LIN {X 0,Y 420.578,Z 342.697,A -85,B 0,C 180,E1 -10184.764,E2 -10184.764} C_VEL
LIN {X 0,Y 421.368,Z 331.394,A -85,B 0,C 180,E1 -10185.603,E2 -10185.603} C_VEL
LIN {X 0,Y 422.106,Z 318.707,A -85,B 0,C 180,E1 -10186.319,E2 -10186.319} C_VEL
LIN {X 0,Y 422.68,Z 306.29,A -85,B 0,C 180,E1 -10186.824,E2 -10186.824} C_VEL
LIN {X 0,Y 423.128,Z 292.678,A -85,B 0,C 180,E1 -10187.179,E2 -10187.179} C_VEL
LIN {X 0,Y 424.249,Z 215.121,A -85,B 0,C 180,E1 -10188.698,E2 -10188.698} C_VEL
LIN {X 0,Y 420.632,Z 193.799,A -85,B 0,C 180,E1 -10189.35,E2 -10189.35} C_VEL
LIN {X 0,Y 419.974,Z 190.079,A -85,B 0,C 180,E1 -10189.487,E2 -10189.487} C_VEL
LIN {X 0,Y 421.119,Z 172.26,A -85,B 0,C 180,E1 -10193.004,E2 -10193.004} C_VEL
LIN {X 0,Y 421.346,Z 166.733,A -85,B 0,C 180,E1 -10194.121,E2 -10194.121} C_VEL
LIN {X 0,Y 419.386,Z 156.606,A -85,B 0,C 180,E1 -10196.365,E2 -10196.365} C_VEL
LIN {X 0,Y 418.209,Z 151.397,A -85,B 0,C 180,E1 -10197.595,E2 -10197.595} C_VEL
LIN {X 0,Y 418.236,Z 151.388,A -85,B 0,C 180,E1 -10200.274,E2 -10200.274} C_VEL
LIN {X 0,Y 418.234,Z 151.388,A -85,B 0,C 180,E1 -10203.679,E2 -10203.679} C_VEL
LIN {X 0,Y 418.236,Z 151.388,A -85,B 0,C 180,E1 -10207.225,E2 -10207.225} C_VEL
LIN {X 0,Y 418.209,Z 151.393,A -85,B 0,C 180,E1 -10210.868,E2 -10210.868} C_VEL
LIN {X 0,Y 418.205,Z 151.387,A -85,B 0,C 180,E1 -10213.729,E2 -10213.729} C_VEL
LIN {X 0,Y 418.203,Z 151.387,A -85,B 0,C 180,E1 -10216.448,E2 -10216.448} C_VEL
LIN {X 0,Y 418.209,Z 151.387,A -85,B 0,C 180,E1 -10219.133,E2 -10219.133} C_VEL
LIN {X 0,Y 418.239,Z 151.388,A -85,B 0,C 180,E1 -10222.776,E2 -10222.776} C_VEL
LIN {X 0,Y 418.236,Z 151.387,A -85,B 0,C 180,E1 -10226.322,E2 -10226.322} C_VEL
LIN {X 0,Y 418.241,Z 151.382,A -85,B 0,C 180,E1 -10229.728,E2 -10229.728} C_VEL
LIN {X 0,Y 418.213,Z 151.388,A -85,B 0,C 180,E1 -10233.017,E2 -10233.017} C_VEL
LIN {X 0,Y 418.262,Z 151.384,A -85,B 0,C 180,E1 -10236.217,E2 -10236.217} C_VEL
LIN {X 0,Y 418.253,Z 151.38,A -85,B 0,C 180,E1 -10239.337,E2 -10239.337} C_VEL
LIN {X 0,Y 418.259,Z 151.387,A -85,B 0,C 180,E1 -10242.395,E2 -10242.395} C_VEL
LIN {X 0,Y 418.283,Z 151.382,A -85,B 0,C 180,E1 -10245.402,E2 -10245.402} C_VEL
LIN {X 0,Y 418.317,Z 151.379,A -85,B 0,C 180,E1 -10248.369,E2 -10248.369} C_VEL
LIN {X 0,Y 418.45,Z 151.364,A -85,B 0,C 180,E1 -10252.278,E2 -10252.278} C_VEL
LIN {X 0,Y 418.488,Z 151.359,A -85,B 0,C 180,E1 -10254.217,E2 -10254.217} C_VEL
LIN {X 0,Y 418.538,Z 151.353,A -85,B 0,C 180,E1 -10258.076,E2 -10258.076} C_VEL
LIN {X 0,Y 418.567,Z 151.351,A -85,B 0,C 180,E1 -10260,E2 -10260} C_VEL
LIN {X 0,Y 418.494,Z 151.36,A -85,B 0,C 180,E1 -10262.888,E2 -10262.888} C_VEL
LIN {X 0,Y 418.322,Z 151.452,A -85,B 0,C 180,E1 -10264.396,E2 -10264.396} C_VEL
LIN {X 0,Y 420.077,Z 159.254,A -85,B 0,C 180,E1 -10266.243,E2 -10266.243} C_VEL
LIN {X 0,Y 420.765,Z 163.432,A -85,B 0,C 180,E1 -10267.197,E2 -10267.197} C_VEL
LIN {X 0,Y 420.544,Z 170.284,A -85,B 0,C 180,E1 -10268.62,E2 -10268.62} C_VEL
LIN {X 0,Y 424.721,Z 189.71,A -85,B 0,C 180,E1 -10269.272,E2 -10269.272} C_VEL
LIN {X 0,Y 423.098,Z 278.42,A -85,B 0,C 180,E1 -10271.027,E2 -10271.027} C_VEL
LIN {X 0,Y 422.665,Z 291.77,A -85,B 0,C 180,E1 -10271.483,E2 -10271.483} C_VEL
LIN {X 0,Y 422.127,Z 303.733,A -85,B 0,C 180,E1 -10272.073,E2 -10272.073} C_VEL
LIN {X 0,Y 421.492,Z 315.941,A -85,B 0,C 180,E1 -10272.887,E2 -10272.887} C_VEL
LIN {X 0,Y 420.728,Z 327.426,A -85,B 0,C 180,E1 -10273.867,E2 -10273.867} C_VEL
LIN {X 0,Y 419.975,Z 337.256,A -85,B 0,C 180,E1 -10274.91,E2 -10274.91} C_VEL
LIN {X 0,Y 419.33,Z 346.043,A -85,B 0,C 180,E1 -10276.054,E2 -10276.054} C_VEL
LIN {X 0,Y 418.676,Z 354.422,A -85,B 0,C 180,E1 -10277.39,E2 -10277.39} C_VEL
LIN {X 0,Y 418.137,Z 361.95,A -85,B 0,C 180,E1 -10278.873,E2 -10278.873} C_VEL
LIN {X 0,Y 417.715,Z 367.293,A -85,B 0,C 180,E1 -10280.177,E2 -10280.177} C_VEL
LIN {X 0,Y 417.418,Z 372.376,A -85,B 0,C 180,E1 -10281.741,E2 -10281.741} C_VEL
LIN {X 0,Y 417.206,Z 376.186,A -85,B 0,C 180,E1 -10283.32,E2 -10283.32} C_VEL
LIN {X 0,Y 416.984,Z 378.805,A -85,B 0,C 180,E1 -10284.921,E2 -10284.921} C_VEL
LIN {X 0,Y 416.845,Z 380.338,A -85,B 0,C 180,E1 -10286.672,E2 -10286.672} C_VEL
LIN {X 0,Y 416.858,Z 380.431,A -85,B 0,C 180,E1 -10288.753,E2 -10288.753} C_VEL
LIN {X 0,Y 416.972,Z 378.732,A -85,B 0,C 180,E1 -10290.727,E2 -10290.727} C_VEL
LIN {X 0,Y 417.085,Z 376.61,A -85,B 0,C 180,E1 -10292.046,E2 -10292.046} C_VEL
LIN {X 0,Y 417.236,Z 372.609,A -85,B 0,C 180,E1 -10293.77,E2 -10293.77} C_VEL
LIN {X 0,Y 417.524,Z 366.971,A -85,B 0,C 180,E1 -10295.502,E2 -10295.502} C_VEL
LIN {X 0,Y 417.854,Z 360.816,A -85,B 0,C 180,E1 -10296.963,E2 -10296.963} C_VEL
LIN {X 0,Y 418.368,Z 353.097,A -85,B 0,C 180,E1 -10298.43,E2 -10298.43} C_VEL
LIN {X 0,Y 418.92,Z 344.378,A -85,B 0,C 180,E1 -10299.763,E2 -10299.763} C_VEL
LIN {X 0,Y 419.513,Z 333.739,A -85,B 0,C 180,E1 -10301.072,E2 -10301.072} C_VEL
LIN {X 0,Y 420.165,Z 323.007,A -85,B 0,C 180,E1 -10302.129,E2 -10302.129} C_VEL
LIN {X 0,Y 420.845,Z 311.186,A -85,B 0,C 180,E1 -10303.044,E2 -10303.044} C_VEL
LIN {X 0,Y 421.385,Z 298.499,A -85,B 0,C 180,E1 -10303.801,E2 -10303.801} C_VEL
LIN {X 0,Y 421.825,Z 285.338,A -85,B 0,C 180,E1 -10304.359,E2 -10304.359} C_VEL
LIN {X 0,Y 422.202,Z 272.242,A -85,B 0,C 180,E1 -10304.714,E2 -10304.714} C_VEL
LIN {X 0,Y 423.374,Z 189.479,A -85,B 0,C 180,E1 -10306.269,E2 -10306.269} C_VEL
LIN {X 0,Y 419.77,Z 169.472,A -85,B 0,C 180,E1 -10306.836,E2 -10306.836} C_VEL
LIN {X 0,Y 420.098,Z 162.133,A -85,B 0,C 180,E1 -10308.499,E2 -10308.499} C_VEL
LIN {X 0,Y 418.696,Z 153.617,A -85,B 0,C 180,E1 -10310.546,E2 -10310.546} C_VEL
LIN {X 0,Y 418.278,Z 151.384,A -85,B 0,C 180,E1 -10311.098,E2 -10311.098} C_VEL
LIN {X 0,Y 418.246,Z 151.387,A -85,B 0,C 180,E1 -10313.975,E2 -10313.975} C_VEL
LIN {X 0,Y 418.254,Z 151.382,A -85,B 0,C 180,E1 -10317.158,E2 -10317.158} C_VEL
LIN {X 0,Y 418.26,Z 151.383,A -85,B 0,C 180,E1 -10320.837,E2 -10320.837} C_VEL
LIN {X 0,Y 418.216,Z 151.39,A -85,B 0,C 180,E1 -10324.092,E2 -10324.092} C_VEL
LIN {X 0,Y 418.237,Z 151.385,A -85,B 0,C 180,E1 -10325.759,E2 -10325.759} C_VEL
LIN {X 0,Y 417.607,Z 151.468,A -85,B 0,C 180,E1 -10326.562,E2 -10326.562} C_VEL
LIN {X 0,Y 414.834,Z 151.81,A -85,B 0,C 180,E1 -10327.868,E2 -10327.868} C_VEL
LIN {X 0,Y 412.43,Z 152.108,A -85,B 0,C 180,E1 -10328.922,E2 -10328.922} C_VEL
LIN {X 0,Y 411.333,Z 152.246,A -85,B 0,C 180,E1 -10329.736,E2 -10329.736} C_VEL
LIN {X 0,Y 411.209,Z 152.264,A -85,B 0,C 180,E1 -10330.012,E2 -10330.012} C_VEL
LIN {X 0,Y 411.224,Z 152.257,A -85,B 0,C 180,E1 -10333.151,E2 -10333.151} C_VEL
LIN {X 0,Y 411.311,Z 152.247,A -85,B 0,C 180,E1 -10336.896,E2 -10336.896} C_VEL
LIN {X 0,Y 411.281,Z 152.255,A -85,B 0,C 180,E1 -10340.16,E2 -10340.16} C_VEL
LIN {X 0,Y 411.395,Z 152.236,A -85,B 0,C 180,E1 -10343.131,E2 -10343.131} C_VEL
LIN {X 0,Y 411.289,Z 152.249,A -85,B 0,C 180,E1 -10345.098,E2 -10345.098} C_VEL
LIN {X 0,Y 411.506,Z 152.227,A -85,B 0,C 180,E1 -10348.042,E2 -10348.042} C_VEL
LIN {X 0,Y 411.38,Z 152.238,A -85,B 0,C 180,E1 -10350.978,E2 -10350.978} C_VEL
LIN {X 0,Y 411.431,Z 152.232,A -85,B 0,C 180,E1 -10352.937,E2 -10352.937} C_VEL
LIN {X 0,Y 411.391,Z 152.237,A -85,B 0,C 180,E1 -10356.867,E2 -10356.867} C_VEL
LIN {X 0,Y 411.279,Z 152.255,A -85,B 0,C 180,E1 -10359.838,E2 -10359.838} C_VEL
LIN {X 0,Y 411.308,Z 152.249,A -85,B 0,C 180,E1 -10363.102,E2 -10363.102} C_VEL
LIN {X 0,Y 411.209,Z 152.26,A -85,B 0,C 180,E1 -10366.89,E2 -10366.89} C_VEL
LIN {X 0,Y 411.205,Z 152.261,A -85,B 0,C 180,E1 -10369.987,E2 -10369.987} C_VEL
LIN {X 0,Y 411.188,Z 152.267,A -85,B 0,C 180,E1 -10373.147,E2 -10373.147} C_VEL
LIN {X 0,Y 411.172,Z 152.264,A -85,B 0,C 180,E1 -10376.384,E2 -10376.384} C_VEL
LIN {X 0,Y 411.194,Z 152.263,A -85,B 0,C 180,E1 -10379.712,E2 -10379.712} C_VEL
LIN {X 0,Y 411.203,Z 152.267,A -85,B 0,C 180,E1 -10383.155,E2 -10383.155} C_VEL
LIN {X 0,Y 411.19,Z 152.263,A -85,B 0,C 180,E1 -10386.551,E2 -10386.551} C_VEL
LIN {X 0,Y 411.175,Z 152.264,A -85,B 0,C 180,E1 -10389.721,E2 -10389.721} C_VEL
LIN {X 0,Y 411.159,Z 152.27,A -85,B 0,C 180,E1 -10393.134,E2 -10393.134} C_VEL
LIN {X 0,Y 411.16,Z 152.265,A -85,B 0,C 180,E1 -10395.881,E2 -10395.881} C_VEL
LIN {X 0,Y 411.154,Z 152.266,A -85,B 0,C 180,E1 -10399.492,E2 -10399.492} C_VEL
LIN {X 0,Y 411.179,Z 152.263,A -85,B 0,C 180,E1 -10402.024,E2 -10402.024} C_VEL
LIN {X 0,Y 411.198,Z 152.263,A -85,B 0,C 180,E1 -10405.122,E2 -10405.122} C_VEL
LIN {X 0,Y 411.158,Z 152.267,A -85,B 0,C 180,E1 -10408.002,E2 -10408.002} C_VEL
LIN {X 0,Y 411.165,Z 152.265,A -85,B 0,C 180,E1 -10411.406,E2 -10411.406} C_VEL
LIN {X 0,Y 411.182,Z 152.264,A -85,B 0,C 180,E1 -10414.94,E2 -10414.94} C_VEL
LIN {X 0,Y 411.195,Z 152.263,A -85,B 0,C 180,E1 -10417.913,E2 -10417.913} C_VEL
LIN {X 0,Y 411.207,Z 152.26,A -85,B 0,C 180,E1 -10421.05,E2 -10421.05} C_VEL
LIN {X 0,Y 411.203,Z 152.265,A -85,B 0,C 180,E1 -10424.129,E2 -10424.129} C_VEL
LIN {X 0,Y 411.295,Z 152.248,A -85,B 0,C 180,E1 -10427.165,E2 -10427.165} C_VEL
LIN {X 0,Y 411.268,Z 152.259,A -85,B 0,C 180,E1 -10430.16,E2 -10430.16} C_VEL
LIN {X 0,Y 411.383,Z 152.237,A -85,B 0,C 180,E1 -10433.131,E2 -10433.131} C_VEL
LIN {X 0,Y 411.281,Z 152.25,A -85,B 0,C 180,E1 -10435.098,E2 -10435.098} C_VEL
LIN {X 0,Y 411.494,Z 152.23,A -85,B 0,C 180,E1 -10438.042,E2 -10438.042} C_VEL
LIN {X 0,Y 411.368,Z 152.239,A -85,B 0,C 180,E1 -10440.979,E2 -10440.979} C_VEL
LIN {X 0,Y 411.419,Z 152.233,A -85,B 0,C 180,E1 -10442.937,E2 -10442.937} C_VEL
LIN {X 0,Y 411.419,Z 152.239,A -85,B 0,C 180,E1 -10445.883,E2 -10445.883} C_VEL
LIN {X 0,Y 411.298,Z 152.248,A -85,B 0,C 180,E1 -10448.846,E2 -10448.846} C_VEL
LIN {X 0,Y 411.266,Z 152.257,A -85,B 0,C 180,E1 -10451.833,E2 -10451.833} C_VEL
LIN {X 0,Y 411.221,Z 152.258,A -85,B 0,C 180,E1 -10454.854,E2 -10454.854} C_VEL
LIN {X 0,Y 411.17,Z 152.267,A -85,B 0,C 180,E1 -10457.919,E2 -10457.919} C_VEL
LIN {X 0,Y 411.178,Z 152.265,A -85,B 0,C 180,E1 -10461.035,E2 -10461.035} C_VEL
LIN {X 0,Y 411.18,Z 152.263,A -85,B 0,C 180,E1 -10464.218,E2 -10464.218} C_VEL
LIN {X 0,Y 411.136,Z 152.274,A -85,B 0,C 180,E1 -10467.486,E2 -10467.486} C_VEL
LIN {X 0,Y 411.185,Z 152.265,A -85,B 0,C 180,E1 -10469.714,E2 -10469.714} C_VEL
LIN {X 0,Y 411.197,Z 152.267,A -85,B 0,C 180,E1 -10473.157,E2 -10473.157} C_VEL
LIN {X 0,Y 411.182,Z 152.263,A -85,B 0,C 180,E1 -10476.552,E2 -10476.552} C_VEL
LIN {X 0,Y 411.161,Z 152.266,A -85,B 0,C 180,E1 -10479.721,E2 -10479.721} C_VEL
LIN {X 0,Y 411.155,Z 152.272,A -85,B 0,C 180,E1 -10483.136,E2 -10483.136} C_VEL
LIN {X 0,Y 411.158,Z 152.265,A -85,B 0,C 180,E1 -10485.883,E2 -10485.883} C_VEL
LIN {X 0,Y 411.153,Z 152.267,A -85,B 0,C 180,E1 -10489.494,E2 -10489.494} C_VEL
LIN {X 0,Y 411.176,Z 152.263,A -85,B 0,C 180,E1 -10492.026,E2 -10492.026} C_VEL
LIN {X 0,Y 411.197,Z 152.264,A -85,B 0,C 180,E1 -10495.124,E2 -10495.124} C_VEL
LIN {X 0,Y 411.155,Z 152.266,A -85,B 0,C 180,E1 -10498.003,E2 -10498.003} C_VEL
LIN {X 0,Y 411.165,Z 152.267,A -85,B 0,C 180,E1 -10501.407,E2 -10501.407} C_VEL
LIN {X 0,Y 411.203,Z 152.471,A -85,B 0,C 180,E1 -10502.716,E2 -10502.716} C_VEL
LIN {X 0,Y 413.85,Z 165.762,A -85,B 0,C 180,E1 -10505.682,E2 -10505.682} C_VEL
LIN {X 0,Y 413.938,Z 170.108,A -85,B 0,C 180,E1 -10506.593,E2 -10506.593} C_VEL
LIN {X 0,Y 413.243,Z 180.993,A -85,B 0,C 180,E1 -10508.815,E2 -10508.815} C_VEL
LIN {X 0,Y 412.56,Z 191.635,A -85,B 0,C 180,E1 -10510.923,E2 -10510.923} C_VEL
LIN {X 0,Y 416.315,Z 216.844,A -85,B 0,C 180,E1 -10511.579,E2 -10511.579} C_VEL
LIN {X 0,Y 415.097,Z 300.369,A -85,B 0,C 180,E1 -10513.21,E2 -10513.21} C_VEL
LIN {X 0,Y 414.541,Z 314.458,A -85,B 0,C 180,E1 -10513.693,E2 -10513.693} C_VEL
LIN {X 0,Y 413.983,Z 326.514,A -85,B 0,C 180,E1 -10514.303,E2 -10514.303} C_VEL
LIN {X 0,Y 413.303,Z 338.276,A -85,B 0,C 180,E1 -10515.097,E2 -10515.097} C_VEL
LIN {X 0,Y 412.61,Z 349.81,A -85,B 0,C 180,E1 -10516.092,E2 -10516.092} C_VEL
LIN {X 0,Y 411.954,Z 359.966,A -85,B 0,C 180,E1 -10517.187,E2 -10517.187} C_VEL
LIN {X 0,Y 411.366,Z 369.225,A -85,B 0,C 180,E1 -10518.42,E2 -10518.42} C_VEL
LIN {X 0,Y 410.821,Z 378.248,A -85,B 0,C 180,E1 -10519.902,E2 -10519.902} C_VEL
LIN {X 0,Y 410.422,Z 385.465,A -85,B 0,C 180,E1 -10521.384,E2 -10521.384} C_VEL
LIN {X 0,Y 410.162,Z 392.029,A -85,B 0,C 180,E1 -10523.112,E2 -10523.112} C_VEL
LIN {X 0,Y 410.011,Z 396.332,A -85,B 0,C 180,E1 -10524.591,E2 -10524.591} C_VEL
LIN {X 0,Y 409.931,Z 399.529,A -85,B 0,C 180,E1 -10526.069,E2 -10526.069} C_VEL
LIN {X 0,Y 409.928,Z 401.113,A -85,B 0,C 180,E1 -10527.053,E2 -10527.053} C_VEL
LIN {X 0,Y 409.966,Z 402.238,A -85,B 0,C 180,E1 -10528.036,E2 -10528.036} C_VEL
LIN {X 0,Y 409.936,Z 402.929,A -85,B 0,C 180,E1 -10529.019,E2 -10529.019} C_VEL
LIN {X 0,Y 409.928,Z 403.22,A -85,B 0,C 180,E1 -10530.001,E2 -10530.001} C_VEL
LIN {X 0,Y 409.936,Z 403.108,A -85,B 0,C 180,E1 -10530.983,E2 -10530.983} C_VEL
LIN {X 0,Y 409.966,Z 402.547,A -85,B 0,C 180,E1 -10531.966,E2 -10531.966} C_VEL
LIN {X 0,Y 409.924,Z 401.57,A -85,B 0,C 180,E1 -10532.949,E2 -10532.949} C_VEL
LIN {X 0,Y 409.931,Z 400.185,A -85,B 0,C 180,E1 -10533.933,E2 -10533.933} C_VEL
LIN {X 0,Y 410.013,Z 397.264,A -85,B 0,C 180,E1 -10535.41,E2 -10535.41} C_VEL
LIN {X 0,Y 410.167,Z 393.284,A -85,B 0,C 180,E1 -10536.89,E2 -10536.89} C_VEL
LIN {X 0,Y 410.467,Z 387.179,A -85,B 0,C 180,E1 -10538.617,E2 -10538.617} C_VEL
LIN {X 0,Y 410.9,Z 380.464,A -85,B 0,C 180,E1 -10540.098,E2 -10540.098} C_VEL
LIN {X 0,Y 411.501,Z 372.131,A -85,B 0,C 180,E1 -10541.577,E2 -10541.577} C_VEL
LIN {X 0,Y 412.262,Z 363.629,A -85,B 0,C 180,E1 -10542.805,E2 -10542.805} C_VEL
LIN {X 0,Y 412.924,Z 353.201,A -85,B 0,C 180,E1 -10544.035,E2 -10544.035} C_VEL
LIN {X 0,Y 413.849,Z 341.458,A -85,B 0,C 180,E1 -10545.136,E2 -10545.136} C_VEL
LIN {X 0,Y 414.691,Z 329.881,A -85,B 0,C 180,E1 -10545.987,E2 -10545.987} C_VEL
LIN {X 0,Y 415.443,Z 316.74,A -85,B 0,C 180,E1 -10546.714,E2 -10546.714} C_VEL
LIN {X 0,Y 416.1,Z 303.661,A -85,B 0,C 180,E1 -10547.225,E2 -10547.225} C_VEL
LIN {X 0,Y 416.513,Z 288.254,A -85,B 0,C 180,E1 -10547.587,E2 -10547.587} C_VEL
LIN {X 0,Y 417.662,Z 216.047,A -85,B 0,C 180,E1 -10549.042,E2 -10549.042} C_VEL
LIN {X 0,Y 413.962,Z 194.236,A -85,B 0,C 180,E1 -10549.727,E2 -10549.727} C_VEL
LIN {X 0,Y 413.153,Z 189.85,A -85,B 0,C 180,E1 -10549.891,E2 -10549.891} C_VEL
LIN {X 0,Y 414.318,Z 172.758,A -85,B 0,C 180,E1 -10553.335,E2 -10553.335} C_VEL
LIN {X 0,Y 414.465,Z 168.182,A -85,B 0,C 180,E1 -10554.281,E2 -10554.281} C_VEL
LIN {X 0,Y 412.487,Z 158.086,A -85,B 0,C 180,E1 -10556.568,E2 -10556.568} C_VEL
LIN {X 0,Y 411.167,Z 152.272,A -85,B 0,C 180,E1 -10557.969,E2 -10557.969} C_VEL
LIN {X 0,Y 411.186,Z 152.269,A -85,B 0,C 180,E1 -10560.849,E2 -10560.849} C_VEL
LIN {X 0,Y 411.194,Z 152.264,A -85,B 0,C 180,E1 -10564.335,E2 -10564.335} C_VEL
LIN {X 0,Y 411.188,Z 152.268,A -85,B 0,C 180,E1 -10566.743,E2 -10566.743} C_VEL
LIN {X 0,Y 411.17,Z 152.267,A -85,B 0,C 180,E1 -10569.721,E2 -10569.721} C_VEL
LIN {X 0,Y 411.165,Z 152.267,A -85,B 0,C 180,E1 -10573.136,E2 -10573.136} C_VEL
LIN {X 0,Y 411.167,Z 152.262,A -85,B 0,C 180,E1 -10575.882,E2 -10575.882} C_VEL
LIN {X 0,Y 411.161,Z 152.264,A -85,B 0,C 180,E1 -10579.493,E2 -10579.493} C_VEL
LIN {X 0,Y 411.187,Z 152.261,A -85,B 0,C 180,E1 -10582.025,E2 -10582.025} C_VEL
LIN {X 0,Y 411.206,Z 152.263,A -85,B 0,C 180,E1 -10585.124,E2 -10585.124} C_VEL
LIN {X 0,Y 411.167,Z 152.268,A -85,B 0,C 180,E1 -10588.003,E2 -10588.003} C_VEL
LIN {X 0,Y 411.174,Z 152.263,A -85,B 0,C 180,E1 -10591.407,E2 -10591.407} C_VEL
LIN {X 0,Y 411.191,Z 152.263,A -85,B 0,C 180,E1 -10594.942,E2 -10594.942} C_VEL
LIN {X 0,Y 411.207,Z 152.262,A -85,B 0,C 180,E1 -10597.914,E2 -10597.914} C_VEL
LIN {X 0,Y 411.218,Z 152.259,A -85,B 0,C 180,E1 -10601.051,E2 -10601.051} C_VEL
LIN {X 0,Y 411.215,Z 152.262,A -85,B 0,C 180,E1 -10604.13,E2 -10604.13} C_VEL
LIN {X 0,Y 411.308,Z 152.251,A -85,B 0,C 180,E1 -10607.166,E2 -10607.166} C_VEL
LIN {X 0,Y 411.292,Z 152.255,A -85,B 0,C 180,E1 -10610.161,E2 -10610.161} C_VEL
LIN {X 0,Y 411.394,Z 152.242,A -85,B 0,C 180,E1 -10613.132,E2 -10613.132} C_VEL
LIN {X 0,Y 411.294,Z 152.253,A -85,B 0,C 180,E1 -10615.099,E2 -10615.099} C_VEL
LIN {X 0,Y 411.506,Z 152.229,A -85,B 0,C 180,E1 -10618.043,E2 -10618.043} C_VEL
LIN {X 0,Y 411.519,Z 152.229,A -85,B 0,C 180,E1 -10620,E2 -10620} C_VEL
LIN {X 0,Y 411.451,Z 152.238,A -85,B 0,C 180,E1 -10622.938,E2 -10622.938} C_VEL
LIN {X 0,Y 411.285,Z 152.396,A -85,B 0,C 180,E1 -10624.042,E2 -10624.042} C_VEL
LIN {X 0,Y 413.244,Z 160.916,A -85,B 0,C 180,E1 -10626.102,E2 -10626.102} C_VEL
LIN {X 0,Y 413.947,Z 166.194,A -85,B 0,C 180,E1 -10627.316,E2 -10627.316} C_VEL
LIN {X 0,Y 413.696,Z 170.425,A -85,B 0,C 180,E1 -10628.211,E2 -10628.211} C_VEL
LIN {X 0,Y 417.966,Z 189.659,A -85,B 0,C 180,E1 -10628.887,E2 -10628.887} C_VEL
LIN {X 0,Y 418.143,Z 194.672,A -85,B 0,C 180,E1 -10629.005,E2 -10629.005} C_VEL
LIN {X 0,Y 416.403,Z 279.017,A -85,B 0,C 180,E1 -10630.718,E2 -10630.718} C_VEL
LIN {X 0,Y 415.943,Z 291.904,A -85,B 0,C 180,E1 -10631.169,E2 -10631.169} C_VEL
LIN {X 0,Y 415.373,Z 304.045,A -85,B 0,C 180,E1 -10631.777,E2 -10631.777} C_VEL
LIN {X 0,Y 414.713,Z 316.222,A -85,B 0,C 180,E1 -10632.603,E2 -10632.603} C_VEL
LIN {X 0,Y 413.893,Z 327.999,A -85,B 0,C 180,E1 -10633.627,E2 -10633.627} C_VEL
LIN {X 0,Y 413.035,Z 338.568,A -85,B 0,C 180,E1 -10634.788,E2 -10634.788} C_VEL
LIN {X 0,Y 412.291,Z 348.029,A -85,B 0,C 180,E1 -10636.082,E2 -10636.082} C_VEL
LIN {X 0,Y 411.633,Z 356.12,A -85,B 0,C 180,E1 -10637.44,E2 -10637.44} C_VEL
LIN {X 0,Y 411.03,Z 363.399,A -85,B 0,C 180,E1 -10638.958,E2 -10638.958} C_VEL
LIN {X 0,Y 410.584,Z 369.364,A -85,B 0,C 180,E1 -10640.543,E2 -10640.543} C_VEL
LIN {X 0,Y 410.248,Z 374.442,A -85,B 0,C 180,E1 -10642.318,E2 -10642.318} C_VEL
LIN {X 0,Y 410.14,Z 376.405,A -85,B 0,C 180,E1 -10643.211,E2 -10643.211} C_VEL
LIN {X 0,Y 409.938,Z 378.827,A -85,B 0,C 180,E1 -10644.681,E2 -10644.681} C_VEL
LIN {X 0,Y 409.758,Z 380.48,A -85,B 0,C 180,E1 -10646.484,E2 -10646.484} C_VEL
LIN {X 0,Y 409.741,Z 380.817,A -85,B 0,C 180,E1 -10647.589,E2 -10647.589} C_VEL
LIN {X 0,Y 409.77,Z 380.491,A -85,B 0,C 180,E1 -10648.989,E2 -10648.989} C_VEL
LIN {X 0,Y 409.915,Z 378.646,A -85,B 0,C 180,E1 -10650.955,E2 -10650.955} C_VEL
LIN {X 0,Y 410.06,Z 375.137,A -85,B 0,C 180,E1 -10652.879,E2 -10652.879} C_VEL
LIN {X 0,Y 410.24,Z 371.051,A -85,B 0,C 180,E1 -10654.426,E2 -10654.426} C_VEL
LIN {X 0,Y 410.553,Z 365.497,A -85,B 0,C 180,E1 -10656.025,E2 -10656.025} C_VEL
LIN {X 0,Y 410.924,Z 359.528,A -85,B 0,C 180,E1 -10657.385,E2 -10657.385} C_VEL
LIN {X 0,Y 411.448,Z 351.162,A -85,B 0,C 180,E1 -10658.912,E2 -10658.912} C_VEL
LIN {X 0,Y 412.038,Z 342.195,A -85,B 0,C 180,E1 -10660.236,E2 -10660.236} C_VEL
LIN {X 0,Y 412.657,Z 331.913,A -85,B 0,C 180,E1 -10661.463,E2 -10661.463} C_VEL
LIN {X 0,Y 413.348,Z 320.8,A -85,B 0,C 180,E1 -10662.521,E2 -10662.521} C_VEL
LIN {X 0,Y 414.024,Z 309.293,A -85,B 0,C 180,E1 -10663.39,E2 -10663.39} C_VEL
LIN {X 0,Y 414.554,Z 296.968,A -85,B 0,C 180,E1 -10664.1,E2 -10664.1} C_VEL
LIN {X 0,Y 414.985,Z 283.337,A -85,B 0,C 180,E1 -10664.659,E2 -10664.659} C_VEL
LIN {X 0,Y 415.364,Z 269.808,A -85,B 0,C 180,E1 -10664.998,E2 -10664.998} C_VEL
LIN {X 0,Y 416.54,Z 190.275,A -85,B 0,C 180,E1 -10666.525,E2 -10666.525} C_VEL
LIN {X 0,Y 412.843,Z 169.677,A -85,B 0,C 180,E1 -10667.112,E2 -10667.112} C_VEL
LIN {X 0,Y 413.086,Z 162.445,A -85,B 0,C 180,E1 -10668.779,E2 -10668.779} C_VEL
LIN {X 0,Y 411.224,Z 152.261,A -85,B 0,C 180,E1 -10671.315,E2 -10671.315} C_VEL
LIN {X 0,Y 411.199,Z 152.267,A -85,B 0,C 180,E1 -10674.47,E2 -10674.47} C_VEL
LIN {X 0,Y 411.211,Z 152.262,A -85,B 0,C 180,E1 -10676.874,E2 -10676.874} C_VEL
LIN {X 0,Y 411.213,Z 152.263,A -85,B 0,C 180,E1 -10680.65,E2 -10680.65} C_VEL
LIN {X 0,Y 411.169,Z 152.264,A -85,B 0,C 180,E1 -10683.614,E2 -10683.614} C_VEL
LIN {X 0,Y 411.19,Z 152.263,A -85,B 0,C 180,E1 -10686.851,E2 -10686.851} C_VEL
LIN {X 0,Y 411.209,Z 152.264,A -85,B 0,C 180,E1 -10690.012,E2 -10690.012} C_VEL
LIN {X 0,Y 410.455,Z 152.364,A -85,B 0,C 180,E1 -10690.83,E2 -10690.83} C_VEL
LIN {X 0,Y 407.602,Z 152.72,A -85,B 0,C 180,E1 -10692.16,E2 -10692.16} C_VEL
LIN {X 0,Y 405.246,Z 153.008,A -85,B 0,C 180,E1 -10693.234,E2 -10693.234} C_VEL
LIN {X 0,Y 404.245,Z 153.133,A -85,B 0,C 180,E1 -10694.064,E2 -10694.064} C_VEL
LIN {X 0,Y 404.165,Z 153.137,A -85,B 0,C 180,E1 -10694.344,E2 -10694.344} C_VEL
LIN {X 0,Y 404.289,Z 153.121,A -85,B 0,C 180,E1 -10696.938,E2 -10696.938} C_VEL
LIN {X 0,Y 404.248,Z 153.133,A -85,B 0,C 180,E1 -10699.987,E2 -10699.987} C_VEL
LIN {X 0,Y 404.345,Z 153.114,A -85,B 0,C 180,E1 -10703.011,E2 -10703.011} C_VEL
LIN {X 0,Y 404.26,Z 153.125,A -85,B 0,C 180,E1 -10705.012,E2 -10705.012} C_VEL
LIN {X 0,Y 404.475,Z 153.103,A -85,B 0,C 180,E1 -10708.008,E2 -10708.008} C_VEL
LIN {X 0,Y 404.351,Z 153.114,A -85,B 0,C 180,E1 -10710.995,E2 -10710.995} C_VEL
LIN {X 0,Y 404.39,Z 153.109,A -85,B 0,C 180,E1 -10712.988,E2 -10712.988} C_VEL
LIN {X 0,Y 404.342,Z 153.115,A -85,B 0,C 180,E1 -10716.988,E2 -10716.988} C_VEL
LIN {X 0,Y 404.246,Z 153.129,A -85,B 0,C 180,E1 -10720.011,E2 -10720.011} C_VEL
LIN {X 0,Y 404.27,Z 153.127,A -85,B 0,C 180,E1 -10723.21,E2 -10723.21} C_VEL
LIN {X 0,Y 404.157,Z 153.14,A -85,B 0,C 180,E1 -10726.977,E2 -10726.977} C_VEL
LIN {X 0,Y 404.152,Z 153.138,A -85,B 0,C 180,E1 -10730.351,E2 -10730.351} C_VEL
LIN {X 0,Y 404.149,Z 153.143,A -85,B 0,C 180,E1 -10733.575,E2 -10733.575} C_VEL
LIN {X 0,Y 404.104,Z 153.147,A -85,B 0,C 180,E1 -10736.883,E2 -10736.883} C_VEL
LIN {X 0,Y 404.14,Z 153.14,A -85,B 0,C 180,E1 -10740.284,E2 -10740.284} C_VEL
LIN {X 0,Y 404.136,Z 153.141,A -85,B 0,C 180,E1 -10743.812,E2 -10743.812} C_VEL
LIN {X 0,Y 404.133,Z 153.146,A -85,B 0,C 180,E1 -10746.873,E2 -10746.873} C_VEL
LIN {X 0,Y 404.114,Z 153.143,A -85,B 0,C 180,E1 -10750.074,E2 -10750.074} C_VEL
LIN {X 0,Y 404.139,Z 153.145,A -85,B 0,C 180,E1 -10753.081,E2 -10753.081} C_VEL
LIN {X 0,Y 404.117,Z 153.142,A -85,B 0,C 180,E1 -10755.921,E2 -10755.921} C_VEL
LIN {X 0,Y 404.098,Z 153.15,A -85,B 0,C 180,E1 -10758.632,E2 -10758.632} C_VEL
LIN {X 0,Y 404.134,Z 153.141,A -85,B 0,C 180,E1 -10761.494,E2 -10761.494} C_VEL
LIN {X 0,Y 404.173,Z 153.139,A -85,B 0,C 180,E1 -10764.982,E2 -10764.982} C_VEL
LIN {X 0,Y 404.132,Z 153.146,A -85,B 0,C 180,E1 -10768.442,E2 -10768.442} C_VEL
LIN {X 0,Y 404.143,Z 153.143,A -85,B 0,C 180,E1 -10770.861,E2 -10770.861} C_VEL
LIN {X 0,Y 404.146,Z 153.143,A -85,B 0,C 180,E1 -10774.722,E2 -10774.722} C_VEL
LIN {X 0,Y 404.159,Z 153.137,A -85,B 0,C 180,E1 -10777.507,E2 -10777.507} C_VEL
LIN {X 0,Y 404.152,Z 153.141,A -85,B 0,C 180,E1 -10780.707,E2 -10780.707} C_VEL
LIN {X 0,Y 404.174,Z 153.138,A -85,B 0,C 180,E1 -10783.846,E2 -10783.846} C_VEL
LIN {X 0,Y 404.276,Z 153.123,A -85,B 0,C 180,E1 -10786.938,E2 -10786.938} C_VEL
LIN {X 0,Y 404.236,Z 153.133,A -85,B 0,C 180,E1 -10789.987,E2 -10789.987} C_VEL
LIN {X 0,Y 404.333,Z 153.116,A -85,B 0,C 180,E1 -10793.011,E2 -10793.011} C_VEL
LIN {X 0,Y 404.252,Z 153.126,A -85,B 0,C 180,E1 -10795.013,E2 -10795.013} C_VEL
LIN {X 0,Y 404.463,Z 153.106,A -85,B 0,C 180,E1 -10798.008,E2 -10798.008} C_VEL
LIN {X 0,Y 404.339,Z 153.115,A -85,B 0,C 180,E1 -10800.996,E2 -10800.996} C_VEL
LIN {X 0,Y 404.379,Z 153.11,A -85,B 0,C 180,E1 -10802.989,E2 -10802.989} C_VEL
LIN {X 0,Y 404.368,Z 153.116,A -85,B 0,C 180,E1 -10805.986,E2 -10805.986} C_VEL
LIN {X 0,Y 404.247,Z 153.127,A -85,B 0,C 180,E1 -10809.002,E2 -10809.002} C_VEL
LIN {X 0,Y 404.241,Z 153.13,A -85,B 0,C 180,E1 -10812.042,E2 -10812.042} C_VEL
LIN {X 0,Y 404.166,Z 153.138,A -85,B 0,C 180,E1 -10815.119,E2 -10815.119} C_VEL
LIN {X 0,Y 404.127,Z 153.142,A -85,B 0,C 180,E1 -10818.242,E2 -10818.242} C_VEL
LIN {X 0,Y 404.122,Z 153.148,A -85,B 0,C 180,E1 -10821.42,E2 -10821.42} C_VEL
LIN {X 0,Y 404.126,Z 153.142,A -85,B 0,C 180,E1 -10824.669,E2 -10824.669} C_VEL
LIN {X 0,Y 404.093,Z 153.146,A -85,B 0,C 180,E1 -10828.007,E2 -10828.007} C_VEL
LIN {X 0,Y 404.132,Z 153.141,A -85,B 0,C 180,E1 -10830.286,E2 -10830.286} C_VEL
LIN {X 0,Y 404.13,Z 153.142,A -85,B 0,C 180,E1 -10833.814,E2 -10833.814} C_VEL
LIN {X 0,Y 404.125,Z 153.145,A -85,B 0,C 180,E1 -10836.874,E2 -10836.874} C_VEL
LIN {X 0,Y 404.111,Z 153.143,A -85,B 0,C 180,E1 -10840.075,E2 -10840.075} C_VEL
LIN {X 0,Y 404.135,Z 153.147,A -85,B 0,C 180,E1 -10843.082,E2 -10843.082} C_VEL
LIN {X 0,Y 404.114,Z 153.143,A -85,B 0,C 180,E1 -10845.923,E2 -10845.923} C_VEL
LIN {X 0,Y 404.096,Z 153.149,A -85,B 0,C 180,E1 -10848.633,E2 -10848.633} C_VEL
LIN {X 0,Y 404.132,Z 153.142,A -85,B 0,C 180,E1 -10851.496,E2 -10851.496} C_VEL
LIN {X 0,Y 404.168,Z 153.141,A -85,B 0,C 180,E1 -10854.983,E2 -10854.983} C_VEL
LIN {X 0,Y 404.13,Z 153.145,A -85,B 0,C 180,E1 -10858.445,E2 -10858.445} C_VEL
LIN {X 0,Y 404.144,Z 153.143,A -85,B 0,C 180,E1 -10860.863,E2 -10860.863} C_VEL
LIN {X 0,Y 404.173,Z 153.268,A -85,B 0,C 180,E1 -10862.476,E2 -10862.476} C_VEL
LIN {X 0,Y 406.804,Z 166.618,A -85,B 0,C 180,E1 -10865.505,E2 -10865.505} C_VEL
LIN {X 0,Y 407.05,Z 169.913,A -85,B 0,C 180,E1 -10866.217,E2 -10866.217} C_VEL
LIN {X 0,Y 406.263,Z 181.857,A -85,B 0,C 180,E1 -10868.699,E2 -10868.699} C_VEL
LIN {X 0,Y 405.589,Z 191.179,A -85,B 0,C 180,E1 -10870.614,E2 -10870.614} C_VEL
LIN {X 0,Y 409.478,Z 218.464,A -85,B 0,C 180,E1 -10871.348,E2 -10871.348} C_VEL
LIN {X 0,Y 408.191,Z 300.429,A -85,B 0,C 180,E1 -10872.982,E2 -10872.982} C_VEL
LIN {X 0,Y 407.607,Z 314.416,A -85,B 0,C 180,E1 -10873.472,E2 -10873.472} C_VEL
LIN {X 0,Y 407.028,Z 326.418,A -85,B 0,C 180,E1 -10874.092,E2 -10874.092} C_VEL
LIN {X 0,Y 406.287,Z 338.955,A -85,B 0,C 180,E1 -10874.962,E2 -10874.962} C_VEL
LIN {X 0,Y 405.597,Z 350.203,A -85,B 0,C 180,E1 -10875.962,E2 -10875.962} C_VEL
LIN {X 0,Y 405.009,Z 359.322,A -85,B 0,C 180,E1 -10876.964,E2 -10876.964} C_VEL
LIN {X 0,Y 404.369,Z 368.668,A -85,B 0,C 180,E1 -10878.217,E2 -10878.217} C_VEL
LIN {X 0,Y 403.765,Z 377.756,A -85,B 0,C 180,E1 -10879.724,E2 -10879.724} C_VEL
LIN {X 0,Y 403.371,Z 385.052,A -85,B 0,C 180,E1 -10881.232,E2 -10881.232} C_VEL
LIN {X 0,Y 403.073,Z 391.666,A -85,B 0,C 180,E1 -10882.99,E2 -10882.99} C_VEL
LIN {X 0,Y 402.909,Z 396.011,A -85,B 0,C 180,E1 -10884.496,E2 -10884.496} C_VEL
LIN {X 0,Y 402.853,Z 399.247,A -85,B 0,C 180,E1 -10885.999,E2 -10885.999} C_VEL
LIN {X 0,Y 402.827,Z 400.847,A -85,B 0,C 180,E1 -10887.001,E2 -10887.001} C_VEL
LIN {X 0,Y 402.879,Z 402.004,A -85,B 0,C 180,E1 -10888.001,E2 -10888.001} C_VEL
LIN {X 0,Y 402.863,Z 402.711,A -85,B 0,C 180,E1 -10889.001,E2 -10889.001} C_VEL
LIN {X 0,Y 402.852,Z 403.015,A -85,B 0,C 180,E1 -10890.001,E2 -10890.001} C_VEL
LIN {X 0,Y 402.863,Z 402.918,A -85,B 0,C 180,E1 -10891,E2 -10891} C_VEL
LIN {X 0,Y 402.864,Z 402.38,A -85,B 0,C 180,E1 -10892,E2 -10892} C_VEL
LIN {X 0,Y 402.823,Z 401.414,A -85,B 0,C 180,E1 -10893.001,E2 -10893.001} C_VEL
LIN {X 0,Y 402.851,Z 400.043,A -85,B 0,C 180,E1 -10894.002,E2 -10894.002} C_VEL
LIN {X 0,Y 402.911,Z 397.147,A -85,B 0,C 180,E1 -10895.506,E2 -10895.506} C_VEL
LIN {X 0,Y 403.08,Z 393.194,A -85,B 0,C 180,E1 -10897.011,E2 -10897.011} C_VEL
LIN {X 0,Y 403.355,Z 388.087,A -85,B 0,C 180,E1 -10898.518,E2 -10898.518} C_VEL
LIN {X 0,Y 403.795,Z 381.677,A -85,B 0,C 180,E1 -10900.024,E2 -10900.024} C_VEL
LIN {X 0,Y 404.394,Z 373.668,A -85,B 0,C 180,E1 -10901.53,E2 -10901.53} C_VEL
LIN {X 0,Y 405.336,Z 363.701,A -85,B 0,C 180,E1 -10903.027,E2 -10903.027} C_VEL
LIN {X 0,Y 405.981,Z 354.06,A -85,B 0,C 180,E1 -10904.205,E2 -10904.205} C_VEL
LIN {X 0,Y 406.881,Z 343.126,A -85,B 0,C 180,E1 -10905.273,E2 -10905.273} C_VEL
LIN {X 0,Y 407.759,Z 332.075,A -85,B 0,C 180,E1 -10906.137,E2 -10906.137} C_VEL
LIN {X 0,Y 408.566,Z 319.941,A -85,B 0,C 180,E1 -10906.875,E2 -10906.875} C_VEL
LIN {X 0,Y 409.221,Z 307.424,A -85,B 0,C 180,E1 -10907.427,E2 -10907.427} C_VEL
LIN {X 0,Y 409.766,Z 293.559,A -85,B 0,C 180,E1 -10907.822,E2 -10907.822} C_VEL
LIN {X 0,Y 411.125,Z 217.146,A -85,B 0,C 180,E1 -10909.392,E2 -10909.392} C_VEL
LIN {X 0,Y 407.818,Z 197.335,A -85,B 0,C 180,E1 -10910.031,E2 -10910.031} C_VEL
LIN {X 0,Y 406.341,Z 189.571,A -85,B 0,C 180,E1 -10910.328,E2 -10910.328} C_VEL
LIN {X 0,Y 407.499,Z 173.719,A -85,B 0,C 180,E1 -10913.585,E2 -10913.585} C_VEL
LIN {X 0,Y 407.579,Z 169.632,A -85,B 0,C 180,E1 -10914.447,E2 -10914.447} C_VEL
LIN {X 0,Y 405.619,Z 159.613,A -85,B 0,C 180,E1 -10916.776,E2 -10916.776} C_VEL
LIN {X 0,Y 404.14,Z 153.147,A -85,B 0,C 180,E1 -10918.358,E2 -10918.358} C_VEL
LIN {X 0,Y 404.136,Z 153.147,A -85,B 0,C 180,E1 -10921.557,E2 -10921.557} C_VEL
LIN {X 0,Y 404.175,Z 153.143,A -85,B 0,C 180,E1 -10925.018,E2 -10925.018} C_VEL
LIN {X 0,Y 404.135,Z 153.147,A -85,B 0,C 180,E1 -10928.76,E2 -10928.76} C_VEL
LIN {X 0,Y 404.109,Z 153.145,A -85,B 0,C 180,E1 -10931.597,E2 -10931.597} C_VEL
LIN {X 0,Y 404.146,Z 153.141,A -85,B 0,C 180,E1 -10934.522,E2 -10934.522} C_VEL
LIN {X 0,Y 404.124,Z 153.142,A -85,B 0,C 180,E1 -10937.294,E2 -10937.294} C_VEL
LIN {X 0,Y 404.136,Z 153.139,A -85,B 0,C 180,E1 -10939.951,E2 -10939.951} C_VEL
LIN {X 0,Y 404.137,Z 153.141,A -85,B 0,C 180,E1 -10943.126,E2 -10943.126} C_VEL
LIN {X 0,Y 404.141,Z 153.143,A -85,B 0,C 180,E1 -10946.187,E2 -10946.187} C_VEL
LIN {X 0,Y 404.145,Z 153.138,A -85,B 0,C 180,E1 -10949.715,E2 -10949.715} C_VEL
LIN {X 0,Y 404.107,Z 153.145,A -85,B 0,C 180,E1 -10953.117,E2 -10953.117} C_VEL
LIN {X 0,Y 404.153,Z 153.139,A -85,B 0,C 180,E1 -10956.425,E2 -10956.425} C_VEL
LIN {X 0,Y 404.195,Z 153.134,A -85,B 0,C 180,E1 -10959.875,E2 -10959.875} C_VEL
LIN {X 0,Y 404.178,Z 153.138,A -85,B 0,C 180,E1 -10963.013,E2 -10963.013} C_VEL
LIN {X 0,Y 404.287,Z 153.125,A -85,B 0,C 180,E1 -10966.939,E2 -10966.939} C_VEL
LIN {X 0,Y 404.258,Z 153.131,A -85,B 0,C 180,E1 -10969.988,E2 -10969.988} C_VEL
LIN {X 0,Y 404.345,Z 153.12,A -85,B 0,C 180,E1 -10973.012,E2 -10973.012} C_VEL
LIN {X 0,Y 404.266,Z 153.129,A -85,B 0,C 180,E1 -10975.014,E2 -10975.014} C_VEL
LIN {X 0,Y 404.475,Z 153.105,A -85,B 0,C 180,E1 -10978.009,E2 -10978.009} C_VEL
LIN {X 0,Y 404.355,Z 153.121,A -85,B 0,C 180,E1 -10980.996,E2 -10980.996} C_VEL
LIN {X 0,Y 404.41,Z 153.116,A -85,B 0,C 180,E1 -10982.989,E2 -10982.989} C_VEL
LIN {X 0,Y 404.266,Z 153.139,A -85,B 0,C 180,E1 -10983.613,E2 -10983.613} C_VEL
LIN {X 0,Y 406.396,Z 162.594,A -85,B 0,C 180,E1 -10985.956,E2 -10985.956} C_VEL
LIN {X 0,Y 407.103,Z 167.867,A -85,B 0,C 180,E1 -10987.19,E2 -10987.19} C_VEL
LIN {X 0,Y 406.933,Z 170.701,A -85,B 0,C 180,E1 -10987.786,E2 -10987.786} C_VEL
LIN {X 0,Y 410.996,Z 188.506,A -85,B 0,C 180,E1 -10988.451,E2 -10988.451} C_VEL
LIN {X 0,Y 411.624,Z 191.798,A -85,B 0,C 180,E1 -10988.561,E2 -10988.561} C_VEL
LIN {X 0,Y 409.744,Z 279.231,A -85,B 0,C 180,E1 -10990.376,E2 -10990.376} C_VEL
LIN {X 0,Y 409.263,Z 292.629,A -85,B 0,C 180,E1 -10990.857,E2 -10990.857} C_VEL
LIN {X 0,Y 408.652,Z 304.827,A -85,B 0,C 180,E1 -10991.49,E2 -10991.49} C_VEL
LIN {X 0,Y 407.934,Z 316.603,A -85,B 0,C 180,E1 -10992.31,E2 -10992.31} C_VEL
LIN {X 0,Y 407.092,Z 328.299,A -85,B 0,C 180,E1 -10993.351,E2 -10993.351} C_VEL
LIN {X 0,Y 406.177,Z 338.633,A -85,B 0,C 180,E1 -10994.503,E2 -10994.503} C_VEL
LIN {X 0,Y 405.364,Z 348.315,A -85,B 0,C 180,E1 -10995.847,E2 -10995.847} C_VEL
LIN {X 0,Y 404.666,Z 356.311,A -85,B 0,C 180,E1 -10997.212,E2 -10997.212} C_VEL
LIN {X 0,Y 404.045,Z 363.66,A -85,B 0,C 180,E1 -10998.772,E2 -10998.772} C_VEL
LIN {X 0,Y 403.541,Z 369.625,A -85,B 0,C 180,E1 -11000.385,E2 -11000.385} C_VEL
LIN {X 0,Y 403.233,Z 374.159,A -85,B 0,C 180,E1 -11001.977,E2 -11001.977} C_VEL
LIN {X 0,Y 402.972,Z 377.631,A -85,B 0,C 180,E1 -11003.649,E2 -11003.649} C_VEL
LIN {X 0,Y 402.825,Z 379.373,A -85,B 0,C 180,E1 -11004.873,E2 -11004.873} C_VEL
LIN {X 0,Y 402.708,Z 380.329,A -85,B 0,C 180,E1 -11005.868,E2 -11005.868} C_VEL
LIN {X 0,Y 402.681,Z 380.959,A -85,B 0,C 180,E1 -11007.112,E2 -11007.112} C_VEL
LIN {X 0,Y 402.661,Z 380.981,A -85,B 0,C 180,E1 -11008.116,E2 -11008.116} C_VEL
LIN {X 0,Y 402.677,Z 380.536,A -85,B 0,C 180,E1 -11009.255,E2 -11009.255} C_VEL
LIN {X 0,Y 402.748,Z 379.511,A -85,B 0,C 180,E1 -11010.402,E2 -11010.402} C_VEL
LIN {X 0,Y 402.915,Z 376.912,A -85,B 0,C 180,E1 -11012.142,E2 -11012.142} C_VEL
LIN {X 0,Y 403.104,Z 372.9,A -85,B 0,C 180,E1 -11013.912,E2 -11013.912} C_VEL
LIN {X 0,Y 403.395,Z 367.193,A -85,B 0,C 180,E1 -11015.708,E2 -11015.708} C_VEL
LIN {X 0,Y 403.742,Z 361.451,A -85,B 0,C 180,E1 -11017.117,E2 -11017.117} C_VEL
LIN {X 0,Y 404.231,Z 354.402,A -85,B 0,C 180,E1 -11018.52,E2 -11018.52} C_VEL
LIN {X 0,Y 404.871,Z 345.488,A -85,B 0,C 180,E1 -11019.962,E2 -11019.962} C_VEL
LIN {X 0,Y 405.437,Z 335.973,A -85,B 0,C 180,E1 -11021.202,E2 -11021.202} C_VEL
LIN {X 0,Y 406.073,Z 325.841,A -85,B 0,C 180,E1 -11022.277,E2 -11022.277} C_VEL
LIN {X 0,Y 406.833,Z 313.968,A -85,B 0,C 180,E1 -11023.283,E2 -11023.283} C_VEL
LIN {X 0,Y 407.456,Z 302.134,A -85,B 0,C 180,E1 -11024.054,E2 -11024.054} C_VEL
LIN {X 0,Y 407.967,Z 288.317,A -85,B 0,C 180,E1 -11024.718,E2 -11024.718} C_VEL
LIN {X 0,Y 408.325,Z 275.749,A -85,B 0,C 180,E1 -11025.114,E2 -11025.114} C_VEL
LIN {X 0,Y 409.737,Z 191.344,A -85,B 0,C 180,E1 -11026.775,E2 -11026.775} C_VEL
LIN {X 0,Y 405.916,Z 169.857,A -85,B 0,C 180,E1 -11027.4,E2 -11027.4} C_VEL
LIN {X 0,Y 406.103,Z 163.536,A -85,B 0,C 180,E1 -11028.88,E2 -11028.88} C_VEL
LIN {X 0,Y 404.201,Z 153.136,A -85,B 0,C 180,E1 -11031.485,E2 -11031.485} C_VEL
LIN {X 0,Y 404.183,Z 153.136,A -85,B 0,C 180,E1 -11034.983,E2 -11034.983} C_VEL
LIN {X 0,Y 404.139,Z 153.147,A -85,B 0,C 180,E1 -11038.443,E2 -11038.443} C_VEL
LIN {X 0,Y 404.152,Z 153.14,A -85,B 0,C 180,E1 -11040.862,E2 -11040.862} C_VEL
LIN {X 0,Y 404.157,Z 153.14,A -85,B 0,C 180,E1 -11044.723,E2 -11044.723} C_VEL
LIN {X 0,Y 404.169,Z 153.136,A -85,B 0,C 180,E1 -11047.507,E2 -11047.507} C_VEL
LIN {X 0,Y 404.139,Z 153.142,A -85,B 0,C 180,E1 -11050.705,E2 -11050.705} C_VEL
LIN {X 0,Y 404.184,Z 153.138,A -85,B 0,C 180,E1 -11053.846,E2 -11053.846} C_VEL
LIN {X 0,Y 404.165,Z 153.137,A -85,B 0,C 180,E1 -11054.344,E2 -11054.344} C_VEL
LIN {X 0,Y 403.502,Z 153.22,A -85,B 0,C 180,E1 -11055.176,E2 -11055.176} C_VEL
LIN {X 0,Y 400.662,Z 153.575,A -85,B 0,C 180,E1 -11056.529,E2 -11056.529} C_VEL
LIN {X 0,Y 398.271,Z 153.873,A -85,B 0,C 180,E1 -11057.622,E2 -11057.622} C_VEL
LIN {X 0,Y 397.263,Z 153.999,A -85,B 0,C 180,E1 -11058.467,E2 -11058.467} C_VEL
LIN {X 0,Y 397.191,Z 154.006,A -85,B 0,C 180,E1 -11058.753,E2 -11058.753} C_VEL
LIN {X 0,Y 397.312,Z 153.995,A -85,B 0,C 180,E1 -11062.132,E2 -11062.132} C_VEL
LIN {X 0,Y 397.232,Z 154,A -85,B 0,C 180,E1 -11064.924,E2 -11064.924} C_VEL
LIN {X 0,Y 397.443,Z 153.979,A -85,B 0,C 180,E1 -11067.972,E2 -11067.972} C_VEL
LIN {X 0,Y 397.444,Z 153.978,A -85,B 0,C 180,E1 -11072.026,E2 -11072.026} C_VEL
LIN {X 0,Y 397.321,Z 153.992,A -85,B 0,C 180,E1 -11076.091,E2 -11076.091} C_VEL
LIN {X 0,Y 397.23,Z 154.003,A -85,B 0,C 180,E1 -11079.161,E2 -11079.161} C_VEL
LIN {X 0,Y 397.217,Z 154.003,A -85,B 0,C 180,E1 -11082.257,E2 -11082.257} C_VEL
LIN {X 0,Y 397.125,Z 154.019,A -85,B 0,C 180,E1 -11085.393,E2 -11085.393} C_VEL
LIN {X 0,Y 397.089,Z 154.018,A -85,B 0,C 180,E1 -11088.576,E2 -11088.576} C_VEL
LIN {X 0,Y 397.091,Z 154.02,A -85,B 0,C 180,E1 -11091.818,E2 -11091.818} C_VEL
LIN {X 0,Y 397.103,Z 154.021,A -85,B 0,C 180,E1 -11095.134,E2 -11095.134} C_VEL
LIN {X 0,Y 397.062,Z 154.022,A -85,B 0,C 180,E1 -11098.547,E2 -11098.547} C_VEL
LIN {X 0,Y 397.076,Z 154.02,A -85,B 0,C 180,E1 -11101.834,E2 -11101.834} C_VEL
LIN {X 0,Y 397.116,Z 154.016,A -85,B 0,C 180,E1 -11104.493,E2 -11104.493} C_VEL
LIN {X 0,Y 397.091,Z 154.018,A -85,B 0,C 180,E1 -11108.275,E2 -11108.275} C_VEL
LIN {X 0,Y 397.049,Z 154.023,A -85,B 0,C 180,E1 -11111.975,E2 -11111.975} C_VEL
LIN {X 0,Y 397.082,Z 154.023,A -85,B 0,C 180,E1 -11115.068,E2 -11115.068} C_VEL
LIN {X 0,Y 397.047,Z 154.023,A -85,B 0,C 180,E1 -11118.023,E2 -11118.023} C_VEL
LIN {X 0,Y 397.086,Z 154.018,A -85,B 0,C 180,E1 -11121.723,E2 -11121.723} C_VEL
LIN {X 0,Y 397.114,Z 154.015,A -85,B 0,C 180,E1 -11125.505,E2 -11125.505} C_VEL
LIN {X 0,Y 397.07,Z 154.022,A -85,B 0,C 180,E1 -11129.116,E2 -11129.116} C_VEL
LIN {X 0,Y 397.056,Z 154.026,A -85,B 0,C 180,E1 -11132.251,E2 -11132.251} C_VEL
LIN {X 0,Y 397.096,Z 154.02,A -85,B 0,C 180,E1 -11134.864,E2 -11134.864} C_VEL
LIN {X 0,Y 397.087,Z 154.023,A -85,B 0,C 180,E1 -11138.181,E2 -11138.181} C_VEL
LIN {X 0,Y 397.107,Z 154.016,A -85,B 0,C 180,E1 -11141.424,E2 -11141.424} C_VEL
LIN {X 0,Y 397.117,Z 154.018,A -85,B 0,C 180,E1 -11144.605,E2 -11144.605} C_VEL
LIN {X 0,Y 397.207,Z 154.005,A -85,B 0,C 180,E1 -11147.741,E2 -11147.741} C_VEL
LIN {X 0,Y 397.219,Z 154.002,A -85,B 0,C 180,E1 -11150.837,E2 -11150.837} C_VEL
LIN {X 0,Y 397.321,Z 153.994,A -85,B 0,C 180,E1 -11153.907,E2 -11153.907} C_VEL
LIN {X 0,Y 397.431,Z 153.982,A -85,B 0,C 180,E1 -11157.973,E2 -11157.973} C_VEL
LIN {X 0,Y 397.31,Z 153.991,A -85,B 0,C 180,E1 -11161.013,E2 -11161.013} C_VEL
LIN {X 0,Y 397.313,Z 153.99,A -85,B 0,C 180,E1 -11163.042,E2 -11163.042} C_VEL
LIN {X 0,Y 397.319,Z 153.993,A -85,B 0,C 180,E1 -11166.092,E2 -11166.092} C_VEL
LIN {X 0,Y 397.219,Z 154.003,A -85,B 0,C 180,E1 -11169.162,E2 -11169.162} C_VEL
LIN {X 0,Y 397.206,Z 154.005,A -85,B 0,C 180,E1 -11172.258,E2 -11172.258} C_VEL
LIN {X 0,Y 397.115,Z 154.019,A -85,B 0,C 180,E1 -11175.394,E2 -11175.394} C_VEL
LIN {X 0,Y 397.079,Z 154.019,A -85,B 0,C 180,E1 -11178.577,E2 -11178.577} C_VEL
LIN {X 0,Y 397.082,Z 154.022,A -85,B 0,C 180,E1 -11181.819,E2 -11181.819} C_VEL
LIN {X 0,Y 397.095,Z 154.021,A -85,B 0,C 180,E1 -11185.136,E2 -11185.136} C_VEL
LIN {X 0,Y 397.053,Z 154.023,A -85,B 0,C 180,E1 -11188.549,E2 -11188.549} C_VEL
LIN {X 0,Y 397.069,Z 154.022,A -85,B 0,C 180,E1 -11191.836,E2 -11191.836} C_VEL
LIN {X 0,Y 397.109,Z 154.016,A -85,B 0,C 180,E1 -11194.495,E2 -11194.495} C_VEL
LIN {X 0,Y 397.083,Z 154.019,A -85,B 0,C 180,E1 -11198.277,E2 -11198.277} C_VEL
LIN {X 0,Y 397.045,Z 154.024,A -85,B 0,C 180,E1 -11201.977,E2 -11201.977} C_VEL
LIN {X 0,Y 397.08,Z 154.025,A -85,B 0,C 180,E1 -11205.07,E2 -11205.07} C_VEL
LIN {X 0,Y 397.045,Z 154.023,A -85,B 0,C 180,E1 -11208.025,E2 -11208.025} C_VEL
LIN {X 0,Y 397.084,Z 154.019,A -85,B 0,C 180,E1 -11211.724,E2 -11211.724} C_VEL
LIN {X 0,Y 397.112,Z 154.016,A -85,B 0,C 180,E1 -11215.507,E2 -11215.507} C_VEL
LIN {X 0,Y 397.069,Z 154.025,A -85,B 0,C 180,E1 -11219.118,E2 -11219.118} C_VEL
LIN {X 0,Y 397.117,Z 154.084,A -85,B 0,C 180,E1 -11222.237,E2 -11222.237} C_VEL
LIN {X 0,Y 399.763,Z 167.513,A -85,B 0,C 180,E1 -11225.336,E2 -11225.336} C_VEL
LIN {X 0,Y 400.082,Z 171.297,A -85,B 0,C 180,E1 -11226.171,E2 -11226.171} C_VEL
LIN {X 0,Y 399.211,Z 183.331,A -85,B 0,C 180,E1 -11228.71,E2 -11228.71} C_VEL
LIN {X 0,Y 398.635,Z 191.119,A -85,B 0,C 180,E1 -11230.33,E2 -11230.33} C_VEL
LIN {X 0,Y 402.649,Z 218.843,A -85,B 0,C 180,E1 -11231.082,E2 -11231.082} C_VEL
LIN {X 0,Y 401.306,Z 300.332,A -85,B 0,C 180,E1 -11232.746,E2 -11232.746} C_VEL
LIN {X 0,Y 400.698,Z 314.265,A -85,B 0,C 180,E1 -11233.245,E2 -11233.245} C_VEL
LIN {X 0,Y 400.047,Z 327.241,A -85,B 0,C 180,E1 -11233.938,E2 -11233.938} C_VEL
LIN {X 0,Y 399.285,Z 339.577,A -85,B 0,C 180,E1 -11234.823,E2 -11234.823} C_VEL
LIN {X 0,Y 398.669,Z 349.381,A -85,B 0,C 180,E1 -11235.713,E2 -11235.713} C_VEL
LIN {X 0,Y 397.974,Z 359.66,A -85,B 0,C 180,E1 -11236.859,E2 -11236.859} C_VEL
LIN {X 0,Y 397.244,Z 369.744,A -85,B 0,C 180,E1 -11238.262,E2 -11238.262} C_VEL
LIN {X 0,Y 396.646,Z 378.612,A -85,B 0,C 180,E1 -11239.795,E2 -11239.795} C_VEL
LIN {X 0,Y 396.248,Z 385.662,A -85,B 0,C 180,E1 -11241.33,E2 -11241.33} C_VEL
LIN {X 0,Y 396.001,Z 391.293,A -85,B 0,C 180,E1 -11242.865,E2 -11242.865} C_VEL
LIN {X 0,Y 395.823,Z 395.19,A -85,B 0,C 180,E1 -11244.199,E2 -11244.199} C_VEL
LIN {X 0,Y 395.779,Z 398.958,A -85,B 0,C 180,E1 -11245.928,E2 -11245.928} C_VEL
LIN {X 0,Y 395.73,Z 400.576,A -85,B 0,C 180,E1 -11246.947,E2 -11246.947} C_VEL
LIN {X 0,Y 395.778,Z 401.765,A -85,B 0,C 180,E1 -11247.966,E2 -11247.966} C_VEL
LIN {X 0,Y 395.792,Z 402.49,A -85,B 0,C 180,E1 -11248.983,E2 -11248.983} C_VEL
LIN {X 0,Y 395.779,Z 402.81,A -85,B 0,C 180,E1 -11250.001,E2 -11250.001} C_VEL
LIN {X 0,Y 395.791,Z 402.728,A -85,B 0,C 180,E1 -11251.018,E2 -11251.018} C_VEL
LIN {X 0,Y 395.761,Z 402.218,A -85,B 0,C 180,E1 -11252.036,E2 -11252.036} C_VEL
LIN {X 0,Y 395.726,Z 401.265,A -85,B 0,C 180,E1 -11253.055,E2 -11253.055} C_VEL
LIN {X 0,Y 395.774,Z 399.906,A -85,B 0,C 180,E1 -11254.074,E2 -11254.074} C_VEL
LIN {X 0,Y 395.825,Z 396.605,A -85,B 0,C 180,E1 -11255.803,E2 -11255.803} C_VEL
LIN {X 0,Y 396.009,Z 393.115,A -85,B 0,C 180,E1 -11257.137,E2 -11257.137} C_VEL
LIN {X 0,Y 396.316,Z 388.041,A -85,B 0,C 180,E1 -11258.67,E2 -11258.67} C_VEL
LIN {X 0,Y 396.798,Z 381.666,A -85,B 0,C 180,E1 -11260.203,E2 -11260.203} C_VEL
LIN {X 0,Y 397.422,Z 373.713,A -85,B 0,C 180,E1 -11261.735,E2 -11261.735} C_VEL
LIN {X 0,Y 398.42,Z 363.815,A -85,B 0,C 180,E1 -11263.258,E2 -11263.258} C_VEL
LIN {X 0,Y 399.162,Z 353.819,A -85,B 0,C 180,E1 -11264.505,E2 -11264.505} C_VEL
LIN {X 0,Y 400.061,Z 343.48,A -85,B 0,C 180,E1 -11265.54,E2 -11265.54} C_VEL
LIN {X 0,Y 400.973,Z 332.556,A -85,B 0,C 180,E1 -11266.418,E2 -11266.418} C_VEL
LIN {X 0,Y 401.8,Z 320.614,A -85,B 0,C 180,E1 -11267.168,E2 -11267.168} C_VEL
LIN {X 0,Y 402.5,Z 308.596,A -85,B 0,C 180,E1 -11267.727,E2 -11267.727} C_VEL
LIN {X 0,Y 403.101,Z 295.547,A -85,B 0,C 180,E1 -11268.126,E2 -11268.126} C_VEL
LIN {X 0,Y 404.622,Z 218.288,A -85,B 0,C 180,E1 -11269.753,E2 -11269.753} C_VEL
LIN {X 0,Y 401.218,Z 197.737,A -85,B 0,C 180,E1 -11270.446,E2 -11270.446} C_VEL
LIN {X 0,Y 399.518,Z 189.318,A -85,B 0,C 180,E1 -11270.785,E2 -11270.785} C_VEL
LIN {X 0,Y 400.672,Z 174.929,A -85,B 0,C 180,E1 -11273.794,E2 -11273.794} C_VEL
LIN {X 0,Y 400.781,Z 171.764,A -85,B 0,C 180,E1 -11274.478,E2 -11274.478} C_VEL
LIN {X 0,Y 399.027,Z 162.394,A -85,B 0,C 180,E1 -11276.688,E2 -11276.688} C_VEL
LIN {X 0,Y 397.115,Z 154.022,A -85,B 0,C 180,E1 -11278.798,E2 -11278.798} C_VEL
LIN {X 0,Y 397.076,Z 154.025,A -85,B 0,C 180,E1 -11282.073,E2 -11282.073} C_VEL
LIN {X 0,Y 397.1,Z 154.02,A -85,B 0,C 180,E1 -11285.499,E2 -11285.499} C_VEL
LIN {X 0,Y 397.094,Z 154.024,A -85,B 0,C 180,E1 -11288.855,E2 -11288.855} C_VEL
LIN {X 0,Y 397.057,Z 154.024,A -85,B 0,C 180,E1 -11292.27,E2 -11292.27} C_VEL
LIN {X 0,Y 397.088,Z 154.02,A -85,B 0,C 180,E1 -11295.07,E2 -11295.07} C_VEL
LIN {X 0,Y 397.054,Z 154.021,A -85,B 0,C 180,E1 -11298.024,E2 -11298.024} C_VEL
LIN {X 0,Y 397.094,Z 154.015,A -85,B 0,C 180,E1 -11301.724,E2 -11301.724} C_VEL
LIN {X 0,Y 397.12,Z 154.016,A -85,B 0,C 180,E1 -11305.506,E2 -11305.506} C_VEL
LIN {X 0,Y 397.079,Z 154.018,A -85,B 0,C 180,E1 -11309.118,E2 -11309.118} C_VEL
LIN {X 0,Y 397.065,Z 154.022,A -85,B 0,C 180,E1 -11312.252,E2 -11312.252} C_VEL
LIN {X 0,Y 397.106,Z 154.018,A -85,B 0,C 180,E1 -11314.865,E2 -11314.865} C_VEL
LIN {X 0,Y 397.099,Z 154.023,A -85,B 0,C 180,E1 -11318.182,E2 -11318.182} C_VEL
LIN {X 0,Y 397.118,Z 154.016,A -85,B 0,C 180,E1 -11321.425,E2 -11321.425} C_VEL
LIN {X 0,Y 397.129,Z 154.018,A -85,B 0,C 180,E1 -11324.606,E2 -11324.606} C_VEL
LIN {X 0,Y 397.223,Z 154.008,A -85,B 0,C 180,E1 -11327.742,E2 -11327.742} C_VEL
LIN {X 0,Y 397.238,Z 154.005,A -85,B 0,C 180,E1 -11330.838,E2 -11330.838} C_VEL
LIN {X 0,Y 397.332,Z 153.995,A -85,B 0,C 180,E1 -11333.908,E2 -11333.908} C_VEL
LIN {X 0,Y 397.444,Z 153.98,A -85,B 0,C 180,E1 -11337.973,E2 -11337.973} C_VEL
LIN {X 0,Y 397.325,Z 153.997,A -85,B 0,C 180,E1 -11341.014,E2 -11341.014} C_VEL
LIN {X 0,Y 397.318,Z 153.999,A -85,B 0,C 180,E1 -11343.169,E2 -11343.169} C_VEL
LIN {X 0,Y 399.758,Z 165.352,A -85,B 0,C 180,E1 -11346.055,E2 -11346.055} C_VEL
LIN {X 0,Y 400.273,Z 169.564,A -85,B 0,C 180,E1 -11347.06,E2 -11347.06} C_VEL
LIN {X 0,Y 400.221,Z 171.101,A -85,B 0,C 180,E1 -11347.346,E2 -11347.346} C_VEL
LIN {X 0,Y 403.968,Z 187.045,A -85,B 0,C 180,E1 -11347.969,E2 -11347.969} C_VEL
LIN {X 0,Y 405.117,Z 193.647,A -85,B 0,C 180,E1 -11348.197,E2 -11348.197} C_VEL
LIN {X 0,Y 403.143,Z 278.932,A -85,B 0,C 180,E1 -11350.008,E2 -11350.008} C_VEL
LIN {X 0,Y 402.62,Z 292.502,A -85,B 0,C 180,E1 -11350.498,E2 -11350.498} C_VEL
LIN {X 0,Y 402.018,Z 303.898,A -85,B 0,C 180,E1 -11351.087,E2 -11351.087} C_VEL
LIN {X 0,Y 401.245,Z 316.168,A -85,B 0,C 180,E1 -11351.935,E2 -11351.935} C_VEL
LIN {X 0,Y 400.39,Z 327.384,A -85,B 0,C 180,E1 -11352.933,E2 -11352.933} C_VEL
LIN {X 0,Y 399.423,Z 338.184,A -85,B 0,C 180,E1 -11354.131,E2 -11354.131} C_VEL
LIN {X 0,Y 398.597,Z 346.938,A -85,B 0,C 180,E1 -11355.336,E2 -11355.336} C_VEL
LIN {X 0,Y 397.755,Z 356.153,A -85,B 0,C 180,E1 -11356.907,E2 -11356.907} C_VEL
LIN {X 0,Y 397.181,Z 362.772,A -85,B 0,C 180,E1 -11358.306,E2 -11358.306} C_VEL
LIN {X 0,Y 396.66,Z 368.065,A -85,B 0,C 180,E1 -11359.673,E2 -11359.673} C_VEL
LIN {X 0,Y 396.277,Z 373.117,A -85,B 0,C 180,E1 -11361.32,E2 -11361.32} C_VEL
LIN {X 0,Y 396.026,Z 376.88,A -85,B 0,C 180,E1 -11362.981,E2 -11362.981} C_VEL
LIN {X 0,Y 395.816,Z 378.722,A -85,B 0,C 180,E1 -11364.104,E2 -11364.104} C_VEL
LIN {X 0,Y 395.693,Z 380.088,A -85,B 0,C 180,E1 -11365.232,E2 -11365.232} C_VEL
LIN {X 0,Y 395.584,Z 380.901,A -85,B 0,C 180,E1 -11366.37,E2 -11366.37} C_VEL
LIN {X 0,Y 395.579,Z 381.223,A -85,B 0,C 180,E1 -11367.512,E2 -11367.512} C_VEL
LIN {X 0,Y 395.599,Z 380.55,A -85,B 0,C 180,E1 -11369.481,E2 -11369.481} C_VEL
LIN {X 0,Y 395.758,Z 378.195,A -85,B 0,C 180,E1 -11371.525,E2 -11371.525} C_VEL
LIN {X 0,Y 395.953,Z 374.334,A -85,B 0,C 180,E1 -11373.463,E2 -11373.463} C_VEL
LIN {X 0,Y 396.232,Z 368.993,A -85,B 0,C 180,E1 -11375.322,E2 -11375.322} C_VEL
LIN {X 0,Y 396.64,Z 362.405,A -85,B 0,C 180,E1 -11377.045,E2 -11377.045} C_VEL
LIN {X 0,Y 397.187,Z 354.921,A -85,B 0,C 180,E1 -11378.582,E2 -11378.582} C_VEL
LIN {X 0,Y 397.779,Z 346.443,A -85,B 0,C 180,E1 -11379.992,E2 -11379.992} C_VEL
LIN {X 0,Y 398.385,Z 337.168,A -85,B 0,C 180,E1 -11381.25,E2 -11381.25} C_VEL
LIN {X 0,Y 399.07,Z 326.433,A -85,B 0,C 180,E1 -11382.422,E2 -11382.422} C_VEL
LIN {X 0,Y 399.859,Z 314.484,A -85,B 0,C 180,E1 -11383.46,E2 -11383.46} C_VEL
LIN {X 0,Y 400.481,Z 303.302,A -85,B 0,C 180,E1 -11384.214,E2 -11384.214} C_VEL
LIN {X 0,Y 401.004,Z 289.878,A -85,B 0,C 180,E1 -11384.886,E2 -11384.886} C_VEL
LIN {X 0,Y 401.414,Z 276.379,A -85,B 0,C 180,E1 -11385.339,E2 -11385.339} C_VEL
LIN {X 0,Y 402.896,Z 191.91,A -85,B 0,C 180,E1 -11387.046,E2 -11387.046} C_VEL
LIN {X 0,Y 398.971,Z 170.028,A -85,B 0,C 180,E1 -11387.697,E2 -11387.697} C_VEL
LIN {X 0,Y 399.086,Z 164.531,A -85,B 0,C 180,E1 -11389.006,E2 -11389.006} C_VEL
LIN {X 0,Y 397.137,Z 154.016,A -85,B 0,C 180,E1 -11391.728,E2 -11391.728} C_VEL
LIN {X 0,Y 397.125,Z 154.014,A -85,B 0,C 180,E1 -11395.506,E2 -11395.506} C_VEL
LIN {X 0,Y 397.078,Z 154.02,A -85,B 0,C 180,E1 -11399.117,E2 -11399.117} C_VEL
LIN {X 0,Y 397.063,Z 154.027,A -85,B 0,C 180,E1 -11402.252,E2 -11402.252} C_VEL
LIN {X 0,Y 397.107,Z 154.017,A -85,B 0,C 180,E1 -11404.864,E2 -11404.864} C_VEL
LIN {X 0,Y 397.095,Z 154.023,A -85,B 0,C 180,E1 -11408.181,E2 -11408.181} C_VEL
LIN {X 0,Y 397.098,Z 154.017,A -85,B 0,C 180,E1 -11411.423,E2 -11411.423} C_VEL
LIN {X 0,Y 397.127,Z 154.015,A -85,B 0,C 180,E1 -11414.605,E2 -11414.605} C_VEL
LIN {X 0,Y 397.219,Z 154.005,A -85,B 0,C 180,E1 -11417.741,E2 -11417.741} C_VEL
LIN {X 0,Y 397.191,Z 154.006,A -85,B 0,C 180,E1 -11418.753,E2 -11418.753} C_VEL
LIN {X 0,Y 396.554,Z 154.089,A -85,B 0,C 180,E1 -11419.6,E2 -11419.6} C_VEL
LIN {X 0,Y 393.732,Z 154.438,A -85,B 0,C 180,E1 -11420.978,E2 -11420.978} C_VEL
LIN {X 0,Y 391.337,Z 154.74,A -85,B 0,C 180,E1 -11422.091,E2 -11422.091} C_VEL
LIN {X 0,Y 390.323,Z 154.861,A -85,B 0,C 180,E1 -11422.951,E2 -11422.951} C_VEL
LIN {X 0,Y 390.248,Z 154.871,A -85,B 0,C 180,E1 -11423.243,E2 -11423.243} C_VEL
LIN {X 0,Y 390.411,Z 154.856,A -85,B 0,C 180,E1 -11427.936,E2 -11427.936} C_VEL
LIN {X 0,Y 390.411,Z 154.853,A -85,B 0,C 180,E1 -11432.062,E2 -11432.062} C_VEL
LIN {X 0,Y 390.277,Z 154.868,A -85,B 0,C 180,E1 -11436.202,E2 -11436.202} C_VEL
LIN {X 0,Y 390.188,Z 154.881,A -85,B 0,C 180,E1 -11439.328,E2 -11439.328} C_VEL
LIN {X 0,Y 390.198,Z 154.882,A -85,B 0,C 180,E1 -11443.437,E2 -11443.437} C_VEL
LIN {X 0,Y 390.073,Z 154.897,A -85,B 0,C 180,E1 -11447.27,E2 -11447.27} C_VEL
LIN {X 0,Y 390.05,Z 154.899,A -85,B 0,C 180,E1 -11451.121,E2 -11451.121} C_VEL
LIN {X 0,Y 390.042,Z 154.896,A -85,B 0,C 180,E1 -11454.482,E2 -11454.482} C_VEL
LIN {X 0,Y 390.015,Z 154.9,A -85,B 0,C 180,E1 -11457.996,E2 -11457.996} C_VEL
LIN {X 0,Y 390.018,Z 154.902,A -85,B 0,C 180,E1 -11461.504,E2 -11461.504} C_VEL
LIN {X 0,Y 390.068,Z 154.898,A -85,B 0,C 180,E1 -11465.207,E2 -11465.207} C_VEL
LIN {X 0,Y 390.057,Z 154.9,A -85,B 0,C 180,E1 -11469.095,E2 -11469.095} C_VEL
LIN {X 0,Y 390.027,Z 154.899,A -85,B 0,C 180,E1 -11472.371,E2 -11472.371} C_VEL
LIN {X 0,Y 390.038,Z 154.898,A -85,B 0,C 180,E1 -11475.353,E2 -11475.353} C_VEL
LIN {X 0,Y 390.011,Z 154.901,A -85,B 0,C 180,E1 -11478.183,E2 -11478.183} C_VEL
LIN {X 0,Y 390.053,Z 154.9,A -85,B 0,C 180,E1 -11480.903,E2 -11480.903} C_VEL
LIN {X 0,Y 390.076,Z 154.897,A -85,B 0,C 180,E1 -11484.792,E2 -11484.792} C_VEL
LIN {X 0,Y 390.016,Z 154.905,A -85,B 0,C 180,E1 -11488.495,E2 -11488.495} C_VEL
LIN {X 0,Y 390.009,Z 154.902,A -85,B 0,C 180,E1 -11492.002,E2 -11492.002} C_VEL
LIN {X 0,Y 390.035,Z 154.897,A -85,B 0,C 180,E1 -11495.516,E2 -11495.516} C_VEL
LIN {X 0,Y 390.046,Z 154.897,A -85,B 0,C 180,E1 -11498.877,E2 -11498.877} C_VEL
LIN {X 0,Y 390.083,Z 154.896,A -85,B 0,C 180,E1 -11502.164,E2 -11502.164} C_VEL
LIN {X 0,Y 390.085,Z 154.891,A -85,B 0,C 180,E1 -11505.39,E2 -11505.39} C_VEL
LIN {X 0,Y 390.16,Z 154.882,A -85,B 0,C 180,E1 -11507.516,E2 -11507.516} C_VEL
LIN {X 0,Y 390.178,Z 154.88,A -85,B 0,C 180,E1 -11510.67,E2 -11510.67} C_VEL
LIN {X 0,Y 390.275,Z 154.871,A -85,B 0,C 180,E1 -11513.797,E2 -11513.797} C_VEL
LIN {X 0,Y 390.399,Z 154.858,A -85,B 0,C 180,E1 -11517.936,E2 -11517.936} C_VEL
LIN {X 0,Y 390.281,Z 154.866,A -85,B 0,C 180,E1 -11521.032,E2 -11521.032} C_VEL
LIN {X 0,Y 390.249,Z 154.87,A -85,B 0,C 180,E1 -11523.097,E2 -11523.097} C_VEL
LIN {X 0,Y 390.273,Z 154.87,A -85,B 0,C 180,E1 -11526.203,E2 -11526.203} C_VEL
LIN {X 0,Y 390.177,Z 154.881,A -85,B 0,C 180,E1 -11529.329,E2 -11529.329} C_VEL
LIN {X 0,Y 390.187,Z 154.882,A -85,B 0,C 180,E1 -11533.438,E2 -11533.438} C_VEL
LIN {X 0,Y 390.063,Z 154.897,A -85,B 0,C 180,E1 -11537.271,E2 -11537.271} C_VEL
LIN {X 0,Y 390.041,Z 154.899,A -85,B 0,C 180,E1 -11541.123,E2 -11541.123} C_VEL
LIN {X 0,Y 390.033,Z 154.897,A -85,B 0,C 180,E1 -11544.484,E2 -11544.484} C_VEL
LIN {X 0,Y 390.008,Z 154.901,A -85,B 0,C 180,E1 -11547.998,E2 -11547.998} C_VEL
LIN {X 0,Y 390.011,Z 154.904,A -85,B 0,C 180,E1 -11551.505,E2 -11551.505} C_VEL
LIN {X 0,Y 390.061,Z 154.9,A -85,B 0,C 180,E1 -11555.209,E2 -11555.209} C_VEL
LIN {X 0,Y 390.05,Z 154.901,A -85,B 0,C 180,E1 -11559.097,E2 -11559.097} C_VEL
LIN {X 0,Y 390.023,Z 154.899,A -85,B 0,C 180,E1 -11562.373,E2 -11562.373} C_VEL
LIN {X 0,Y 390.035,Z 154.9,A -85,B 0,C 180,E1 -11565.355,E2 -11565.355} C_VEL
LIN {X 0,Y 390.009,Z 154.9,A -85,B 0,C 180,E1 -11568.185,E2 -11568.185} C_VEL
LIN {X 0,Y 390.052,Z 154.901,A -85,B 0,C 180,E1 -11570.904,E2 -11570.904} C_VEL
LIN {X 0,Y 390.064,Z 154.9,A -85,B 0,C 180,E1 -11574.792,E2 -11574.792} C_VEL
LIN {X 0,Y 390.015,Z 154.903,A -85,B 0,C 180,E1 -11578.496,E2 -11578.496} C_VEL
LIN {X 0,Y 390.044,Z 154.935,A -85,B 0,C 180,E1 -11581.995,E2 -11581.995} C_VEL
LIN {X 0,Y 392.692,Z 168.263,A -85,B 0,C 180,E1 -11585.13,E2 -11585.13} C_VEL
LIN {X 0,Y 393.14,Z 171.675,A -85,B 0,C 180,E1 -11585.906,E2 -11585.906} C_VEL
LIN {X 0,Y 392.289,Z 183.279,A -85,B 0,C 180,E1 -11588.402,E2 -11588.402} C_VEL
LIN {X 0,Y 391.725,Z 190.791,A -85,B 0,C 180,E1 -11590.002,E2 -11590.002} C_VEL
LIN {X 0,Y 395.802,Z 219.706,A -85,B 0,C 180,E1 -11590.824,E2 -11590.824} C_VEL
LIN {X 0,Y 394.423,Z 300.153,A -85,B 0,C 180,E1 -11592.502,E2 -11592.502} C_VEL
LIN {X 0,Y 393.786,Z 314.06,A -85,B 0,C 180,E1 -11593.008,E2 -11593.008} C_VEL
LIN {X 0,Y 393.171,Z 326.046,A -85,B 0,C 180,E1 -11593.649,E2 -11593.649} C_VEL
LIN {X 0,Y 392.357,Z 338.576,A -85,B 0,C 180,E1 -11594.548,E2 -11594.548} C_VEL
LIN {X 0,Y 391.635,Z 350.131,A -85,B 0,C 180,E1 -11595.614,E2 -11595.614} C_VEL
LIN {X 0,Y 390.94,Z 359.963,A -85,B 0,C 180,E1 -11596.75,E2 -11596.75} C_VEL
LIN {X 0,Y 390.254,Z 369.142,A -85,B 0,C 180,E1 -11598.048,E2 -11598.048} C_VEL
LIN {X 0,Y 389.597,Z 378.096,A -85,B 0,C 180,E1 -11599.608,E2 -11599.608} C_VEL
LIN {X 0,Y 389.201,Z 385.224,A -85,B 0,C 180,E1 -11601.172,E2 -11601.172} C_VEL
LIN {X 0,Y 388.93,Z 390.907,A -85,B 0,C 180,E1 -11602.734,E2 -11602.734} C_VEL
LIN {X 0,Y 388.724,Z 395.237,A -85,B 0,C 180,E1 -11604.251,E2 -11604.251} C_VEL
LIN {X 0,Y 388.708,Z 398.663,A -85,B 0,C 180,E1 -11605.854,E2 -11605.854} C_VEL
LIN {X 0,Y 388.638,Z 400.3,A -85,B 0,C 180,E1 -11606.891,E2 -11606.891} C_VEL
LIN {X 0,Y 388.676,Z 401.517,A -85,B 0,C 180,E1 -11607.928,E2 -11607.928} C_VEL
LIN {X 0,Y 388.704,Z 402.267,A -85,B 0,C 180,E1 -11608.965,E2 -11608.965} C_VEL
LIN {X 0,Y 388.709,Z 402.603,A -85,B 0,C 180,E1 -11610.001,E2 -11610.001} C_VEL
LIN {X 0,Y 388.703,Z 402.537,A -85,B 0,C 180,E1 -11611.037,E2 -11611.037} C_VEL
LIN {X 0,Y 388.659,Z 402.056,A -85,B 0,C 180,E1 -11612.073,E2 -11612.073} C_VEL
LIN {X 0,Y 388.633,Z 401.121,A -85,B 0,C 180,E1 -11613.111,E2 -11613.111} C_VEL
LIN {X 0,Y 388.698,Z 399.778,A -85,B 0,C 180,E1 -11614.148,E2 -11614.148} C_VEL
LIN {X 0,Y 388.726,Z 396.843,A -85,B 0,C 180,E1 -11615.752,E2 -11615.752} C_VEL
LIN {X 0,Y 388.938,Z 393.046,A -85,B 0,C 180,E1 -11617.268,E2 -11617.268} C_VEL
LIN {X 0,Y 389.29,Z 388.013,A -85,B 0,C 180,E1 -11618.828,E2 -11618.828} C_VEL
LIN {X 0,Y 389.785,Z 381.689,A -85,B 0,C 180,E1 -11620.388,E2 -11620.388} C_VEL
LIN {X 0,Y 390.468,Z 373.822,A -85,B 0,C 180,E1 -11621.947,E2 -11621.947} C_VEL
LIN {X 0,Y 391.51,Z 363.974,A -85,B 0,C 180,E1 -11623.496,E2 -11623.496} C_VEL
LIN {X 0,Y 392.286,Z 354.064,A -85,B 0,C 180,E1 -11624.765,E2 -11624.765} C_VEL
LIN {X 0,Y 393.242,Z 343.835,A -85,B 0,C 180,E1 -11625.817,E2 -11625.817} C_VEL
LIN {X 0,Y 394.35,Z 331.281,A -85,B 0,C 180,E1 -11626.835,E2 -11626.835} C_VEL
LIN {X 0,Y 395.221,Z 319.025,A -85,B 0,C 180,E1 -11627.597,E2 -11627.597} C_VEL
LIN {X 0,Y 395.976,Z 306.338,A -85,B 0,C 180,E1 -11628.163,E2 -11628.163} C_VEL
LIN {X 0,Y 396.562,Z 292.341,A -85,B 0,C 180,E1 -11628.57,E2 -11628.57} C_VEL
LIN {X 0,Y 398.097,Z 219.015,A -85,B 0,C 180,E1 -11630.153,E2 -11630.153} C_VEL
LIN {X 0,Y 394.629,Z 198.263,A -85,B 0,C 180,E1 -11630.875,E2 -11630.875} C_VEL
LIN {X 0,Y 392.717,Z 189.039,A -85,B 0,C 180,E1 -11631.267,E2 -11631.267} C_VEL
LIN {X 0,Y 393.947,Z 175.202,A -85,B 0,C 180,E1 -11634.226,E2 -11634.226} C_VEL
LIN {X 0,Y 393.441,Z 170.179,A -85,B 0,C 180,E1 -11635.387,E2 -11635.387} C_VEL
LIN {X 0,Y 390.95,Z 158.65,A -85,B 0,C 180,E1 -11638.254,E2 -11638.254} C_VEL
LIN {X 0,Y 390.077,Z 154.898,A -85,B 0,C 180,E1 -11639.257,E2 -11639.257} C_VEL
LIN {X 0,Y 390.042,Z 154.901,A -85,B 0,C 180,E1 -11642.722,E2 -11642.722} C_VEL
LIN {X 0,Y 390.044,Z 154.899,A -85,B 0,C 180,E1 -11645.823,E2 -11645.823} C_VEL
LIN {X 0,Y 390.039,Z 154.902,A -85,B 0,C 180,E1 -11649.213,E2 -11649.213} C_VEL
LIN {X 0,Y 390.033,Z 154.899,A -85,B 0,C 180,E1 -11652.372,E2 -11652.372} C_VEL
LIN {X 0,Y 390.044,Z 154.895,A -85,B 0,C 180,E1 -11655.354,E2 -11655.354} C_VEL
LIN {X 0,Y 390.018,Z 154.899,A -85,B 0,C 180,E1 -11658.185,E2 -11658.185} C_VEL
LIN {X 0,Y 390.06,Z 154.892,A -85,B 0,C 180,E1 -11660.904,E2 -11660.904} C_VEL
LIN {X 0,Y 390.072,Z 154.897,A -85,B 0,C 180,E1 -11664.792,E2 -11664.792} C_VEL
LIN {X 0,Y 390.025,Z 154.901,A -85,B 0,C 180,E1 -11668.496,E2 -11668.496} C_VEL
LIN {X 0,Y 390.018,Z 154.898,A -85,B 0,C 180,E1 -11672.003,E2 -11672.003} C_VEL
LIN {X 0,Y 390.046,Z 154.896,A -85,B 0,C 180,E1 -11675.517,E2 -11675.517} C_VEL
LIN {X 0,Y 390.059,Z 154.892,A -85,B 0,C 180,E1 -11678.878,E2 -11678.878} C_VEL
LIN {X 0,Y 390.093,Z 154.893,A -85,B 0,C 180,E1 -11682.165,E2 -11682.165} C_VEL
LIN {X 0,Y 390.096,Z 154.893,A -85,B 0,C 180,E1 -11685.391,E2 -11685.391} C_VEL
LIN {X 0,Y 390.175,Z 154.885,A -85,B 0,C 180,E1 -11687.517,E2 -11687.517} C_VEL
LIN {X 0,Y 390.196,Z 154.883,A -85,B 0,C 180,E1 -11690.671,E2 -11690.671} C_VEL
LIN {X 0,Y 390.287,Z 154.872,A -85,B 0,C 180,E1 -11693.798,E2 -11693.798} C_VEL
LIN {X 0,Y 390.411,Z 154.856,A -85,B 0,C 180,E1 -11697.937,E2 -11697.937} C_VEL
LIN {X 0,Y 390.296,Z 154.873,A -85,B 0,C 180,E1 -11701.032,E2 -11701.032} C_VEL
LIN {X 0,Y 390.357,Z 155.003,A -85,B 0,C 180,E1 -11702.774,E2 -11702.774} C_VEL
LIN {X 0,Y 392.955,Z 167.106,A -85,B 0,C 180,E1 -11705.903,E2 -11705.903} C_VEL
LIN {X 0,Y 393.455,Z 171.033,A -85,B 0,C 180,E1 -11706.861,E2 -11706.861} C_VEL
LIN {X 0,Y 397.375,Z 187.53,A -85,B 0,C 180,E1 -11707.543,E2 -11707.543} C_VEL
LIN {X 0,Y 398.661,Z 194.405,A -85,B 0,C 180,E1 -11707.792,E2 -11707.792} C_VEL
LIN {X 0,Y 396.512,Z 279.983,A -85,B 0,C 180,E1 -11709.662,E2 -11709.662} C_VEL
LIN {X 0,Y 395.977,Z 293.193,A -85,B 0,C 180,E1 -11710.159,E2 -11710.159} C_VEL
LIN {X 0,Y 395.256,Z 305.522,A -85,B 0,C 180,E1 -11710.825,E2 -11710.825} C_VEL
LIN {X 0,Y 394.44,Z 317.553,A -85,B 0,C 180,E1 -11711.697,E2 -11711.697} C_VEL
LIN {X 0,Y 393.497,Z 329.148,A -85,B 0,C 180,E1 -11712.769,E2 -11712.769} C_VEL
LIN {X 0,Y 392.469,Z 339.609,A -85,B 0,C 180,E1 -11713.99,E2 -11713.99} C_VEL
LIN {X 0,Y 391.576,Z 348.844,A -85,B 0,C 180,E1 -11715.325,E2 -11715.325} C_VEL
LIN {X 0,Y 390.798,Z 356.741,A -85,B 0,C 180,E1 -11716.723,E2 -11716.723} C_VEL
LIN {X 0,Y 390.068,Z 364.241,A -85,B 0,C 180,E1 -11718.38,E2 -11718.38} C_VEL
LIN {X 0,Y 389.463,Z 370.697,A -85,B 0,C 180,E1 -11720.22,E2 -11720.22} C_VEL
LIN {X 0,Y 389.123,Z 374.744,A -85,B 0,C 180,E1 -11721.732,E2 -11721.732} C_VEL
LIN {X 0,Y 388.862,Z 378.103,A -85,B 0,C 180,E1 -11723.429,E2 -11723.429} C_VEL
LIN {X 0,Y 388.598,Z 380.418,A -85,B 0,C 180,E1 -11725.272,E2 -11725.272} C_VEL
LIN {X 0,Y 388.506,Z 381.35,A -85,B 0,C 180,E1 -11726.888,E2 -11726.888} C_VEL
LIN {X 0,Y 388.471,Z 381.372,A -85,B 0,C 180,E1 -11728.059,E2 -11728.059} C_VEL
LIN {X 0,Y 388.525,Z 380.511,A -85,B 0,C 180,E1 -11729.741,E2 -11729.741} C_VEL
LIN {X 0,Y 388.705,Z 377.95,A -85,B 0,C 180,E1 -11731.81,E2 -11731.81} C_VEL
LIN {X 0,Y 388.915,Z 373.862,A -85,B 0,C 180,E1 -11733.771,E2 -11733.771} C_VEL
LIN {X 0,Y 389.221,Z 368.317,A -85,B 0,C 180,E1 -11735.653,E2 -11735.653} C_VEL
LIN {X 0,Y 389.624,Z 362.12,A -85,B 0,C 180,E1 -11737.252,E2 -11737.252} C_VEL
LIN {X 0,Y 390.173,Z 354.874,A -85,B 0,C 180,E1 -11738.751,E2 -11738.751} C_VEL
LIN {X 0,Y 390.716,Z 347.214,A -85,B 0,C 180,E1 -11740.051,E2 -11740.051} C_VEL
LIN {X 0,Y 391.404,Z 337.139,A -85,B 0,C 180,E1 -11741.447,E2 -11741.447} C_VEL
LIN {X 0,Y 392.135,Z 326.353,A -85,B 0,C 180,E1 -11742.639,E2 -11742.639} C_VEL
LIN {X 0,Y 392.954,Z 314.325,A -85,B 0,C 180,E1 -11743.695,E2 -11743.695} C_VEL
LIN {X 0,Y 393.607,Z 302.433,A -85,B 0,C 180,E1 -11744.496,E2 -11744.496} C_VEL
LIN {X 0,Y 394.152,Z 288.921,A -85,B 0,C 180,E1 -11745.169,E2 -11745.169} C_VEL
LIN {X 0,Y 394.519,Z 276.601,A -85,B 0,C 180,E1 -11745.58,E2 -11745.58} C_VEL
LIN {X 0,Y 396.104,Z 193.216,A -85,B 0,C 180,E1 -11747.3,E2 -11747.3} C_VEL
LIN {X 0,Y 392.049,Z 170.216,A -85,B 0,C 180,E1 -11747.997,E2 -11747.997} C_VEL
LIN {X 0,Y 391.975,Z 164.859,A -85,B 0,C 180,E1 -11749.302,E2 -11749.302} C_VEL
LIN {X 0,Y 390.087,Z 154.895,A -85,B 0,C 180,E1 -11751.897,E2 -11751.897} C_VEL
LIN {X 0,Y 390.087,Z 154.894,A -85,B 0,C 180,E1 -11754.792,E2 -11754.792} C_VEL
LIN {X 0,Y 390.024,Z 154.905,A -85,B 0,C 180,E1 -11758.495,E2 -11758.495} C_VEL
LIN {X 0,Y 390.02,Z 154.901,A -85,B 0,C 180,E1 -11762.003,E2 -11762.003} C_VEL
LIN {X 0,Y 390.046,Z 154.896,A -85,B 0,C 180,E1 -11765.516,E2 -11765.516} C_VEL
LIN {X 0,Y 390.054,Z 154.895,A -85,B 0,C 180,E1 -11768.877,E2 -11768.877} C_VEL
LIN {X 0,Y 390.059,Z 154.901,A -85,B 0,C 180,E1 -11772.163,E2 -11772.163} C_VEL
LIN {X 0,Y 390.096,Z 154.89,A -85,B 0,C 180,E1 -11775.39,E2 -11775.39} C_VEL
LIN {X 0,Y 390.172,Z 154.881,A -85,B 0,C 180,E1 -11777.516,E2 -11777.516} C_VEL
LIN {X 0,Y 390.19,Z 154.878,A -85,B 0,C 180,E1 -11780.67,E2 -11780.67} C_VEL
LIN {X 0,Y 390.248,Z 154.871,A -85,B 0,C 180,E1 -11783.243,E2 -11783.243} C_VEL
LIN {X 0,Y 389.585,Z 154.958,A -85,B 0,C 180,E1 -11784.103,E2 -11784.103} C_VEL
LIN {X 0,Y 386.694,Z 155.315,A -85,B 0,C 180,E1 -11785.5,E2 -11785.5} C_VEL
LIN {X 0,Y 384.306,Z 155.611,A -85,B 0,C 180,E1 -11786.63,E2 -11786.63} C_VEL
LIN {X 0,Y 383.378,Z 155.729,A -85,B 0,C 180,E1 -11787.504,E2 -11787.504} C_VEL
LIN {X 0,Y 383.354,Z 155.734,A -85,B 0,C 180,E1 -11787.799,E2 -11787.799} C_VEL
LIN {X 0,Y 383.264,Z 155.741,A -85,B 0,C 180,E1 -11791.05,E2 -11791.05} C_VEL
LIN {X 0,Y 383.377,Z 155.729,A -85,B 0,C 180,E1 -11792.1,E2 -11792.1} C_VEL
LIN {X 0,Y 383.235,Z 155.745,A -85,B 0,C 180,E1 -11796.316,E2 -11796.316} C_VEL
LIN {X 0,Y 383.139,Z 155.761,A -85,B 0,C 180,E1 -11799.501,E2 -11799.501} C_VEL
LIN {X 0,Y 383.128,Z 155.764,A -85,B 0,C 180,E1 -11803.535,E2 -11803.535} C_VEL
LIN {X 0,Y 383.026,Z 155.777,A -85,B 0,C 180,E1 -11807.419,E2 -11807.419} C_VEL
LIN {X 0,Y 383.015,Z 155.772,A -85,B 0,C 180,E1 -11810.639,E2 -11810.639} C_VEL
LIN {X 0,Y 383.008,Z 155.774,A -85,B 0,C 180,E1 -11813.808,E2 -11813.808} C_VEL
LIN {X 0,Y 382.969,Z 155.783,A -85,B 0,C 180,E1 -11817.308,E2 -11817.308} C_VEL
LIN {X 0,Y 382.979,Z 155.78,A -85,B 0,C 180,E1 -11820.918,E2 -11820.918} C_VEL
LIN {X 0,Y 383.01,Z 155.774,A -85,B 0,C 180,E1 -11824.667,E2 -11824.667} C_VEL
LIN {X 0,Y 382.992,Z 155.774,A -85,B 0,C 180,E1 -11827.901,E2 -11827.901} C_VEL
LIN {X 0,Y 382.958,Z 155.781,A -85,B 0,C 180,E1 -11831.349,E2 -11831.349} C_VEL
LIN {X 0,Y 382.986,Z 155.776,A -85,B 0,C 180,E1 -11834.301,E2 -11834.301} C_VEL
LIN {X 0,Y 382.993,Z 155.776,A -85,B 0,C 180,E1 -11837.237,E2 -11837.237} C_VEL
LIN {X 0,Y 382.981,Z 155.778,A -85,B 0,C 180,E1 -11840.418,E2 -11840.418} C_VEL
LIN {X 0,Y 383.018,Z 155.772,A -85,B 0,C 180,E1 -11844.043,E2 -11844.043} C_VEL
LIN {X 0,Y 382.98,Z 155.776,A -85,B 0,C 180,E1 -11847.578,E2 -11847.578} C_VEL
LIN {X 0,Y 382.97,Z 155.781,A -85,B 0,C 180,E1 -11850.298,E2 -11850.298} C_VEL
LIN {X 0,Y 382.996,Z 155.776,A -85,B 0,C 180,E1 -11854.044,E2 -11854.044} C_VEL
LIN {X 0,Y 382.979,Z 155.776,A -85,B 0,C 180,E1 -11857.333,E2 -11857.333} C_VEL
LIN {X 0,Y 383.027,Z 155.773,A -85,B 0,C 180,E1 -11860.714,E2 -11860.714} C_VEL
LIN {X 0,Y 383.013,Z 155.775,A -85,B 0,C 180,E1 -11864.023,E2 -11864.023} C_VEL
LIN {X 0,Y 383.127,Z 155.757,A -85,B 0,C 180,E1 -11867.283,E2 -11867.283} C_VEL
LIN {X 0,Y 383.129,Z 155.76,A -85,B 0,C 180,E1 -11870.497,E2 -11870.497} C_VEL
LIN {X 0,Y 383.231,Z 155.747,A -85,B 0,C 180,E1 -11873.683,E2 -11873.683} C_VEL
LIN {X 0,Y 383.365,Z 155.734,A -85,B 0,C 180,E1 -11877.899,E2 -11877.899} C_VEL
LIN {X 0,Y 383.252,Z 155.742,A -85,B 0,C 180,E1 -11881.051,E2 -11881.051} C_VEL
LIN {X 0,Y 383.364,Z 155.732,A -85,B 0,C 180,E1 -11882.101,E2 -11882.101} C_VEL
LIN {X 0,Y 383.23,Z 155.746,A -85,B 0,C 180,E1 -11886.317,E2 -11886.317} C_VEL
LIN {X 0,Y 383.128,Z 155.761,A -85,B 0,C 180,E1 -11889.502,E2 -11889.502} C_VEL
LIN {X 0,Y 383.118,Z 155.764,A -85,B 0,C 180,E1 -11893.536,E2 -11893.536} C_VEL
LIN {X 0,Y 383.016,Z 155.776,A -85,B 0,C 180,E1 -11897.421,E2 -11897.421} C_VEL
LIN {X 0,Y 383.005,Z 155.773,A -85,B 0,C 180,E1 -11900.641,E2 -11900.641} C_VEL
LIN {X 0,Y 382.999,Z 155.776,A -85,B 0,C 180,E1 -11903.809,E2 -11903.809} C_VEL
LIN {X 0,Y 382.96,Z 155.784,A -85,B 0,C 180,E1 -11907.309,E2 -11907.309} C_VEL
LIN {X 0,Y 382.971,Z 155.779,A -85,B 0,C 180,E1 -11910.92,E2 -11910.92} C_VEL
LIN {X 0,Y 383.004,Z 155.774,A -85,B 0,C 180,E1 -11914.669,E2 -11914.669} C_VEL
LIN {X 0,Y 382.985,Z 155.775,A -85,B 0,C 180,E1 -11917.903,E2 -11917.903} C_VEL
LIN {X 0,Y 382.954,Z 155.783,A -85,B 0,C 180,E1 -11921.351,E2 -11921.351} C_VEL
LIN {X 0,Y 382.983,Z 155.776,A -85,B 0,C 180,E1 -11924.303,E2 -11924.303} C_VEL
LIN {X 0,Y 382.976,Z 155.78,A -85,B 0,C 180,E1 -11927.237,E2 -11927.237} C_VEL
LIN {X 0,Y 382.98,Z 155.778,A -85,B 0,C 180,E1 -11930.42,E2 -11930.42} C_VEL
LIN {X 0,Y 383.008,Z 155.772,A -85,B 0,C 180,E1 -11934.044,E2 -11934.044} C_VEL
LIN {X 0,Y 382.979,Z 155.776,A -85,B 0,C 180,E1 -11937.58,E2 -11937.58} C_VEL
LIN {X 0,Y 382.971,Z 155.78,A -85,B 0,C 180,E1 -11940.3,E2 -11940.3} C_VEL
LIN {X 0,Y 382.981,Z 155.778,A -85,B 0,C 180,E1 -11941.744,E2 -11941.744} C_VEL
LIN {X 0,Y 385.353,Z 167.743,A -85,B 0,C 180,E1 -11944.623,E2 -11944.623} C_VEL
LIN {X 0,Y 386.058,Z 171.637,A -85,B 0,C 180,E1 -11945.537,E2 -11945.537} C_VEL
LIN {X 0,Y 385.483,Z 181.792,A -85,B 0,C 180,E1 -11947.772,E2 -11947.772} C_VEL
LIN {X 0,Y 384.822,Z 190.74,A -85,B 0,C 180,E1 -11949.717,E2 -11949.717} C_VEL
LIN {X 0,Y 388.972,Z 220.08,A -85,B 0,C 180,E1 -11950.549,E2 -11950.549} C_VEL
LIN {X 0,Y 387.525,Z 299.742,A -85,B 0,C 180,E1 -11952.249,E2 -11952.249} C_VEL
LIN {X 0,Y 386.88,Z 313.692,A -85,B 0,C 180,E1 -11952.764,E2 -11952.764} C_VEL
LIN {X 0,Y 386.251,Z 325.733,A -85,B 0,C 180,E1 -11953.416,E2 -11953.416} C_VEL
LIN {X 0,Y 385.498,Z 337.497,A -85,B 0,C 180,E1 -11954.266,E2 -11954.266} C_VEL
LIN {X 0,Y 384.698,Z 349.241,A -85,B 0,C 180,E1 -11955.351,E2 -11955.351} C_VEL
LIN {X 0,Y 384.006,Z 359.226,A -85,B 0,C 180,E1 -11956.507,E2 -11956.507} C_VEL
LIN {X 0,Y 383.278,Z 368.498,A -85,B 0,C 180,E1 -11957.828,E2 -11957.828} C_VEL
LIN {X 0,Y 382.55,Z 377.533,A -85,B 0,C 180,E1 -11959.415,E2 -11959.415} C_VEL
LIN {X 0,Y 382.153,Z 384.76,A -85,B 0,C 180,E1 -11961.008,E2 -11961.008} C_VEL
LIN {X 0,Y 381.854,Z 390.501,A -85,B 0,C 180,E1 -11962.599,E2 -11962.599} C_VEL
LIN {X 0,Y 381.625,Z 395.268,A -85,B 0,C 180,E1 -11964.304,E2 -11964.304} C_VEL
LIN {X 0,Y 381.638,Z 398.356,A -85,B 0,C 180,E1 -11965.777,E2 -11965.777} C_VEL
LIN {X 0,Y 381.549,Z 400.013,A -85,B 0,C 180,E1 -11966.833,E2 -11966.833} C_VEL
LIN {X 0,Y 381.575,Z 401.255,A -85,B 0,C 180,E1 -11967.89,E2 -11967.89} C_VEL
LIN {X 0,Y 381.619,Z 402.04,A -85,B 0,C 180,E1 -11968.946,E2 -11968.946} C_VEL
LIN {X 0,Y 381.64,Z 402.396,A -85,B 0,C 180,E1 -11970.001,E2 -11970.001} C_VEL
LIN {X 0,Y 381.603,Z 402.346,A -85,B 0,C 180,E1 -11971.056,E2 -11971.056} C_VEL
LIN {X 0,Y 381.557,Z 401.89,A -85,B 0,C 180,E1 -11972.112,E2 -11972.112} C_VEL
LIN {X 0,Y 381.545,Z 400.982,A -85,B 0,C 180,E1 -11973.169,E2 -11973.169} C_VEL
LIN {X 0,Y 381.623,Z 399.656,A -85,B 0,C 180,E1 -11974.225,E2 -11974.225} C_VEL
LIN {X 0,Y 381.67,Z 396.267,A -85,B 0,C 180,E1 -11976.094,E2 -11976.094} C_VEL
LIN {X 0,Y 381.984,Z 391.495,A -85,B 0,C 180,E1 -11977.932,E2 -11977.932} C_VEL
LIN {X 0,Y 382.479,Z 385.045,A -85,B 0,C 180,E1 -11979.787,E2 -11979.787} C_VEL
LIN {X 0,Y 383.063,Z 378.035,A -85,B 0,C 180,E1 -11981.376,E2 -11981.376} C_VEL
LIN {X 0,Y 384.064,Z 369.299,A -85,B 0,C 180,E1 -11982.955,E2 -11982.955} C_VEL
LIN {X 0,Y 385.005,Z 358.997,A -85,B 0,C 180,E1 -11984.451,E2 -11984.451} C_VEL
LIN {X 0,Y 386.044,Z 348.129,A -85,B 0,C 180,E1 -11985.713,E2 -11985.713} C_VEL
LIN {X 0,Y 387.152,Z 336.87,A -85,B 0,C 180,E1 -11986.75,E2 -11986.75} C_VEL
LIN {X 0,Y 388.2,Z 324.338,A -85,B 0,C 180,E1 -11987.653,E2 -11987.653} C_VEL
LIN {X 0,Y 389.038,Z 311.625,A -85,B 0,C 180,E1 -11988.328,E2 -11988.328} C_VEL
LIN {X 0,Y 389.807,Z 298.582,A -85,B 0,C 180,E1 -11988.801,E2 -11988.801} C_VEL
LIN {X 0,Y 391.579,Z 219.573,A -85,B 0,C 180,E1 -11990.571,E2 -11990.571} C_VEL
LIN {X 0,Y 388.207,Z 199.322,A -85,B 0,C 180,E1 -11991.306,E2 -11991.306} C_VEL
LIN {X 0,Y 385.969,Z 188.934,A -85,B 0,C 180,E1 -11991.74,E2 -11991.74} C_VEL
LIN {X 0,Y 387.128,Z 176.741,A -85,B 0,C 180,E1 -11994.395,E2 -11994.395} C_VEL
LIN {X 0,Y 386.589,Z 171.762,A -85,B 0,C 180,E1 -11995.58,E2 -11995.58} C_VEL
LIN {X 0,Y 384.044,Z 160.116,A -85,B 0,C 180,E1 -11998.55,E2 -11998.55} C_VEL
LIN {X 0,Y 383.045,Z 155.773,A -85,B 0,C 180,E1 -11999.755,E2 -11999.755} C_VEL
LIN {X 0,Y 383.001,Z 155.779,A -85,B 0,C 180,E1 -12003.402,E2 -12003.402} C_VEL
LIN {X 0,Y 383.024,Z 155.774,A -85,B 0,C 180,E1 -12006.163,E2 -12006.163} C_VEL
LIN {X 0,Y 382.988,Z 155.778,A -85,B 0,C 180,E1 -12009.581,E2 -12009.581} C_VEL
LIN {X 0,Y 383.009,Z 155.775,A -85,B 0,C 180,E1 -12012.779,E2 -12012.779} C_VEL
LIN {X 0,Y 382.993,Z 155.772,A -85,B 0,C 180,E1 -12015.789,E2 -12015.789} C_VEL
LIN {X 0,Y 382.964,Z 155.775,A -85,B 0,C 180,E1 -12018.801,E2 -12018.801} C_VEL
LIN {X 0,Y 382.996,Z 155.772,A -85,B 0,C 180,E1 -12022.098,E2 -12022.098} C_VEL
LIN {X 0,Y 383.015,Z 155.774,A -85,B 0,C 180,E1 -12025.332,E2 -12025.332} C_VEL
LIN {X 0,Y 382.984,Z 155.774,A -85,B 0,C 180,E1 -12029.082,E2 -12029.082} C_VEL
LIN {X 0,Y 382.972,Z 155.781,A -85,B 0,C 180,E1 -12032.692,E2 -12032.692} C_VEL
LIN {X 0,Y 383.013,Z 155.774,A -85,B 0,C 180,E1 -12036.191,E2 -12036.191} C_VEL
LIN {X 0,Y 383.06,Z 155.764,A -85,B 0,C 180,E1 -12039.599,E2 -12039.599} C_VEL
LIN {X 0,Y 383.073,Z 155.767,A -85,B 0,C 180,E1 -12042.93,E2 -12042.93} C_VEL
LIN {X 0,Y 383.13,Z 155.761,A -85,B 0,C 180,E1 -12046.464,E2 -12046.464} C_VEL
LIN {X 0,Y 383.146,Z 155.762,A -85,B 0,C 180,E1 -12050.498,E2 -12050.498} C_VEL
LIN {X 0,Y 383.243,Z 155.749,A -85,B 0,C 180,E1 -12053.683,E2 -12053.683} C_VEL
LIN {X 0,Y 383.377,Z 155.732,A -85,B 0,C 180,E1 -12057.899,E2 -12057.899} C_VEL
LIN {X 0,Y 383.267,Z 155.749,A -85,B 0,C 180,E1 -12061.051,E2 -12061.051} C_VEL
LIN {X 0,Y 383.377,Z 155.893,A -85,B 0,C 180,E1 -12062.298,E2 -12062.298} C_VEL
LIN {X 0,Y 386.132,Z 168.895,A -85,B 0,C 180,E1 -12065.746,E2 -12065.746} C_VEL
LIN {X 0,Y 386.544,Z 171.29,A -85,B 0,C 180,E1 -12066.352,E2 -12066.352} C_VEL
LIN {X 0,Y 389.296,Z 181.274,A -85,B 0,C 180,E1 -12066.816,E2 -12066.816} C_VEL
LIN {X 0,Y 392.212,Z 195.773,A -85,B 0,C 180,E1 -12067.388,E2 -12067.388} C_VEL
LIN {X 0,Y 389.97,Z 280.191,A -85,B 0,C 180,E1 -12069.271,E2 -12069.271} C_VEL
LIN {X 0,Y 389.363,Z 293.43,A -85,B 0,C 180,E1 -12069.775,E2 -12069.775} C_VEL
LIN {X 0,Y 388.614,Z 306.209,A -85,B 0,C 180,E1 -12070.485,E2 -12070.485} C_VEL
LIN {X 0,Y 387.737,Z 318.085,A -85,B 0,C 180,E1 -12071.369,E2 -12071.369} C_VEL
LIN {X 0,Y 386.723,Z 329.628,A -85,B 0,C 180,E1 -12072.463,E2 -12072.463} C_VEL
LIN {X 0,Y 385.638,Z 340.01,A -85,B 0,C 180,E1 -12073.705,E2 -12073.705} C_VEL
LIN {X 0,Y 384.689,Z 349.378,A -85,B 0,C 180,E1 -12075.09,E2 -12075.09} C_VEL
LIN {X 0,Y 383.889,Z 357.083,A -85,B 0,C 180,E1 -12076.485,E2 -12076.485} C_VEL
LIN {X 0,Y 383.092,Z 364.563,A -85,B 0,C 180,E1 -12078.172,E2 -12078.172} C_VEL
LIN {X 0,Y 382.474,Z 370.385,A -85,B 0,C 180,E1 -12079.844,E2 -12079.844} C_VEL
LIN {X 0,Y 382.078,Z 375.031,A -85,B 0,C 180,E1 -12081.586,E2 -12081.586} C_VEL
LIN {X 0,Y 381.834,Z 377.883,A -85,B 0,C 180,E1 -12083.029,E2 -12083.029} C_VEL
LIN {X 0,Y 381.516,Z 380.547,A -85,B 0,C 180,E1 -12085.068,E2 -12085.068} C_VEL
LIN {X 0,Y 381.431,Z 381.327,A -85,B 0,C 180,E1 -12086.245,E2 -12086.245} C_VEL
LIN {X 0,Y 381.403,Z 381.607,A -85,B 0,C 180,E1 -12087.811,E2 -12087.811} C_VEL
LIN {X 0,Y 381.437,Z 380.613,A -85,B 0,C 180,E1 -12089.834,E2 -12089.834} C_VEL
LIN {X 0,Y 381.509,Z 379.281,A -85,B 0,C 180,E1 -12091.052,E2 -12091.052} C_VEL
LIN {X 0,Y 381.73,Z 376.133,A -85,B 0,C 180,E1 -12092.897,E2 -12092.897} C_VEL
LIN {X 0,Y 381.951,Z 371.483,A -85,B 0,C 180,E1 -12094.779,E2 -12094.779} C_VEL
LIN {X 0,Y 382.31,Z 366.289,A -85,B 0,C 180,E1 -12096.36,E2 -12096.36} C_VEL
LIN {X 0,Y 382.751,Z 360.136,A -85,B 0,C 180,E1 -12097.855,E2 -12097.855} C_VEL
LIN {X 0,Y 383.337,Z 351.942,A -85,B 0,C 180,E1 -12099.451,E2 -12099.451} C_VEL
LIN {X 0,Y 384.014,Z 342.982,A -85,B 0,C 180,E1 -12100.865,E2 -12100.865} C_VEL
LIN {X 0,Y 384.67,Z 333.724,A -85,B 0,C 180,E1 -12102.062,E2 -12102.062} C_VEL
LIN {X 0,Y 385.485,Z 322.3,A -85,B 0,C 180,E1 -12103.245,E2 -12103.245} C_VEL
LIN {X 0,Y 386.372,Z 309.655,A -85,B 0,C 180,E1 -12104.27,E2 -12104.27} C_VEL
LIN {X 0,Y 386.918,Z 298.008,A -85,B 0,C 180,E1 -12104.988,E2 -12104.988} C_VEL
LIN {X 0,Y 387.424,Z 284.597,A -85,B 0,C 180,E1 -12105.585,E2 -12105.585} C_VEL
LIN {X 0,Y 387.837,Z 271.994,A -85,B 0,C 180,E1 -12105.941,E2 -12105.941} C_VEL
LIN {X 0,Y 389.162,Z 193.305,A -85,B 0,C 180,E1 -12107.594,E2 -12107.594} C_VEL
LIN {X 0,Y 385.125,Z 170.342,A -85,B 0,C 180,E1 -12108.317,E2 -12108.317} C_VEL
LIN {X 0,Y 385.038,Z 166.514,A -85,B 0,C 180,E1 -12109.266,E2 -12109.266} C_VEL
LIN {X 0,Y 383.036,Z 155.774,A -85,B 0,C 180,E1 -12112.09,E2 -12112.09} C_VEL
LIN {X 0,Y 383.023,Z 155.77,A -85,B 0,C 180,E1 -12115.66,E2 -12115.66} C_VEL
LIN {X 0,Y 382.984,Z 155.776,A -85,B 0,C 180,E1 -12119.081,E2 -12119.081} C_VEL
LIN {X 0,Y 382.971,Z 155.78,A -85,B 0,C 180,E1 -12122.691,E2 -12122.691} C_VEL
LIN {X 0,Y 383.012,Z 155.777,A -85,B 0,C 180,E1 -12126.19,E2 -12126.19} C_VEL
LIN {X 0,Y 383.041,Z 155.769,A -85,B 0,C 180,E1 -12129.597,E2 -12129.597} C_VEL
LIN {X 0,Y 383.046,Z 155.768,A -85,B 0,C 180,E1 -12132.928,E2 -12132.928} C_VEL
LIN {X 0,Y 383.131,Z 155.76,A -85,B 0,C 180,E1 -12136.463,E2 -12136.463} C_VEL
LIN {X 0,Y 383.141,Z 155.757,A -85,B 0,C 180,E1 -12140.497,E2 -12140.497} C_VEL
LIN {X 0,Y 383.238,Z 155.747,A -85,B 0,C 180,E1 -12143.682,E2 -12143.682} C_VEL
LIN {X 0,Y 383.354,Z 155.734,A -85,B 0,C 180,E1 -12147.799,E2 -12147.799} C_VEL
LIN {X 0,Y 382.844,Z 155.805,A -85,B 0,C 180,E1 -12148.675,E2 -12148.675} C_VEL
LIN {X 0,Y 380.08,Z 156.151,A -85,B 0,C 180,E1 -12150.1,E2 -12150.1} C_VEL
LIN {X 0,Y 377.584,Z 156.455,A -85,B 0,C 180,E1 -12151.25,E2 -12151.25} C_VEL
LIN {X 0,Y 376.413,Z 156.597,A -85,B 0,C 180,E1 -12152.14,E2 -12152.14} C_VEL
LIN {X 0,Y 376.27,Z 156.612,A -85,B 0,C 180,E1 -12152.443,E2 -12152.443} C_VEL
LIN {X 0,Y 376.195,Z 156.621,A -85,B 0,C 180,E1 -12156.435,E2 -12156.435} C_VEL
LIN {X 0,Y 376.11,Z 156.637,A -85,B 0,C 180,E1 -12159.681,E2 -12159.681} C_VEL
LIN {X 0,Y 376.092,Z 156.639,A -85,B 0,C 180,E1 -12163.656,E2 -12163.656} C_VEL
LIN {X 0,Y 375.984,Z 156.652,A -85,B 0,C 180,E1 -12167.576,E2 -12167.576} C_VEL
LIN {X 0,Y 375.98,Z 156.649,A -85,B 0,C 180,E1 -12170.831,E2 -12170.831} C_VEL
LIN {X 0,Y 375.935,Z 156.653,A -85,B 0,C 180,E1 -12174.284,E2 -12174.284} C_VEL
LIN {X 0,Y 375.911,Z 156.657,A -85,B 0,C 180,E1 -12176.659,E2 -12176.659} C_VEL
LIN {X 0,Y 375.913,Z 156.661,A -85,B 0,C 180,E1 -12179.083,E2 -12179.083} C_VEL
LIN {X 0,Y 375.954,Z 156.653,A -85,B 0,C 180,E1 -12181.561,E2 -12181.561} C_VEL
LIN {X 0,Y 375.948,Z 156.655,A -85,B 0,C 180,E1 -12185.415,E2 -12185.415} C_VEL
LIN {X 0,Y 375.935,Z 156.654,A -85,B 0,C 180,E1 -12188.262,E2 -12188.262} C_VEL
LIN {X 0,Y 375.914,Z 156.657,A -85,B 0,C 180,E1 -12191.596,E2 -12191.596} C_VEL
LIN {X 0,Y 375.918,Z 156.66,A -85,B 0,C 180,E1 -12194.729,E2 -12194.729} C_VEL
LIN {X 0,Y 375.912,Z 156.656,A -85,B 0,C 180,E1 -12197.696,E2 -12197.696} C_VEL
LIN {X 0,Y 375.93,Z 156.658,A -85,B 0,C 180,E1 -12200.533,E2 -12200.533} C_VEL
LIN {X 0,Y 375.957,Z 156.651,A -85,B 0,C 180,E1 -12203.495,E2 -12203.495} C_VEL
LIN {X 0,Y 375.954,Z 156.651,A -85,B 0,C 180,E1 -12205.887,E2 -12205.887} C_VEL
LIN {X 0,Y 375.955,Z 156.651,A -85,B 0,C 180,E1 -12209.686,E2 -12209.686} C_VEL
LIN {X 0,Y 375.911,Z 156.659,A -85,B 0,C 180,E1 -12212.134,E2 -12212.134} C_VEL
LIN {X 0,Y 375.93,Z 156.66,A -85,B 0,C 180,E1 -12214.533,E2 -12214.533} C_VEL
LIN {X 0,Y 375.964,Z 156.652,A -85,B 0,C 180,E1 -12216.886,E2 -12216.886} C_VEL
LIN {X 0,Y 375.969,Z 156.656,A -85,B 0,C 180,E1 -12220.337,E2 -12220.337} C_VEL
LIN {X 0,Y 375.968,Z 156.65,A -85,B 0,C 180,E1 -12223.716,E2 -12223.716} C_VEL
LIN {X 0,Y 376.095,Z 156.633,A -85,B 0,C 180,E1 -12227.041,E2 -12227.041} C_VEL
LIN {X 0,Y 376.1,Z 156.637,A -85,B 0,C 180,E1 -12230.318,E2 -12230.318} C_VEL
LIN {X 0,Y 376.19,Z 156.623,A -85,B 0,C 180,E1 -12233.564,E2 -12233.564} C_VEL
LIN {X 0,Y 376.329,Z 156.609,A -85,B 0,C 180,E1 -12237.859,E2 -12237.859} C_VEL
LIN {X 0,Y 376.223,Z 156.618,A -85,B 0,C 180,E1 -12241.07,E2 -12241.07} C_VEL
LIN {X 0,Y 376.329,Z 156.608,A -85,B 0,C 180,E1 -12242.14,E2 -12242.14} C_VEL
LIN {X 0,Y 376.189,Z 156.623,A -85,B 0,C 180,E1 -12246.436,E2 -12246.436} C_VEL
LIN {X 0,Y 376.099,Z 156.639,A -85,B 0,C 180,E1 -12249.682,E2 -12249.682} C_VEL
LIN {X 0,Y 376.082,Z 156.642,A -85,B 0,C 180,E1 -12253.657,E2 -12253.657} C_VEL
LIN {X 0,Y 375.974,Z 156.655,A -85,B 0,C 180,E1 -12257.577,E2 -12257.577} C_VEL
LIN {X 0,Y 375.971,Z 156.649,A -85,B 0,C 180,E1 -12260.832,E2 -12260.832} C_VEL
LIN {X 0,Y 375.926,Z 156.654,A -85,B 0,C 180,E1 -12264.286,E2 -12264.286} C_VEL
LIN {X 0,Y 375.903,Z 156.658,A -85,B 0,C 180,E1 -12266.661,E2 -12266.661} C_VEL
LIN {X 0,Y 375.905,Z 156.661,A -85,B 0,C 180,E1 -12269.085,E2 -12269.085} C_VEL
LIN {X 0,Y 375.947,Z 156.655,A -85,B 0,C 180,E1 -12271.563,E2 -12271.563} C_VEL
LIN {X 0,Y 375.942,Z 156.657,A -85,B 0,C 180,E1 -12275.417,E2 -12275.417} C_VEL
LIN {X 0,Y 375.927,Z 156.654,A -85,B 0,C 180,E1 -12278.263,E2 -12278.263} C_VEL
LIN {X 0,Y 375.907,Z 156.658,A -85,B 0,C 180,E1 -12281.598,E2 -12281.598} C_VEL
LIN {X 0,Y 375.915,Z 156.659,A -85,B 0,C 180,E1 -12284.731,E2 -12284.731} C_VEL
LIN {X 0,Y 375.902,Z 156.658,A -85,B 0,C 180,E1 -12287.697,E2 -12287.697} C_VEL
LIN {X 0,Y 375.929,Z 156.657,A -85,B 0,C 180,E1 -12290.535,E2 -12290.535} C_VEL
LIN {X 0,Y 375.952,Z 156.652,A -85,B 0,C 180,E1 -12293.498,E2 -12293.498} C_VEL
LIN {X 0,Y 375.953,Z 156.651,A -85,B 0,C 180,E1 -12295.889,E2 -12295.889} C_VEL
LIN {X 0,Y 375.956,Z 156.653,A -85,B 0,C 180,E1 -12299.688,E2 -12299.688} C_VEL
LIN {X 0,Y 375.962,Z 156.788,A -85,B 0,C 180,E1 -12301.536,E2 -12301.536} C_VEL
LIN {X 0,Y 378.277,Z 168.512,A -85,B 0,C 180,E1 -12304.409,E2 -12304.409} C_VEL
LIN {X 0,Y 379.105,Z 173.62,A -85,B 0,C 180,E1 -12305.626,E2 -12305.626} C_VEL
LIN {X 0,Y 378.428,Z 183.834,A -85,B 0,C 180,E1 -12307.91,E2 -12307.91} C_VEL
LIN {X 0,Y 377.858,Z 190.563,A -85,B 0,C 180,E1 -12309.397,E2 -12309.397} C_VEL
LIN {X 0,Y 382.136,Z 221.194,A -85,B 0,C 180,E1 -12310.286,E2 -12310.286} C_VEL
LIN {X 0,Y 380.652,Z 299.24,A -85,B 0,C 180,E1 -12311.987,E2 -12311.987} C_VEL
LIN {X 0,Y 380.008,Z 313.261,A -85,B 0,C 180,E1 -12312.511,E2 -12312.511} C_VEL
LIN {X 0,Y 379.344,Z 325.368,A -85,B 0,C 180,E1 -12313.174,E2 -12313.174} C_VEL
LIN {X 0,Y 378.507,Z 337.96,A -85,B 0,C 180,E1 -12314.106,E2 -12314.106} C_VEL
LIN {X 0,Y 377.683,Z 349.435,A -85,B 0,C 180,E1 -12315.195,E2 -12315.195} C_VEL
LIN {X 0,Y 376.979,Z 359.453,A -85,B 0,C 180,E1 -12316.388,E2 -12316.388} C_VEL
LIN {X 0,Y 376.142,Z 369.492,A -85,B 0,C 180,E1 -12317.867,E2 -12317.867} C_VEL
LIN {X 0,Y 375.515,Z 376.949,A -85,B 0,C 180,E1 -12319.214,E2 -12319.214} C_VEL
LIN {X 0,Y 375.077,Z 384.276,A -85,B 0,C 180,E1 -12320.837,E2 -12320.837} C_VEL
LIN {X 0,Y 374.768,Z 390.082,A -85,B 0,C 180,E1 -12322.458,E2 -12322.458} C_VEL
LIN {X 0,Y 374.582,Z 394.286,A -85,B 0,C 180,E1 -12323.934,E2 -12323.934} C_VEL
LIN {X 0,Y 374.567,Z 398.041,A -85,B 0,C 180,E1 -12325.697,E2 -12325.697} C_VEL
LIN {X 0,Y 374.464,Z 399.72,A -85,B 0,C 180,E1 -12326.773,E2 -12326.773} C_VEL
LIN {X 0,Y 374.475,Z 400.983,A -85,B 0,C 180,E1 -12327.85,E2 -12327.85} C_VEL
LIN {X 0,Y 374.52,Z 401.81,A -85,B 0,C 180,E1 -12328.926,E2 -12328.926} C_VEL
LIN {X 0,Y 374.555,Z 402.186,A -85,B 0,C 180,E1 -12330.001,E2 -12330.001} C_VEL
LIN {X 0,Y 374.503,Z 402.156,A -85,B 0,C 180,E1 -12331.076,E2 -12331.076} C_VEL
LIN {X 0,Y 374.456,Z 401.723,A -85,B 0,C 180,E1 -12332.152,E2 -12332.152} C_VEL
LIN {X 0,Y 374.46,Z 400.853,A -85,B 0,C 180,E1 -12333.229,E2 -12333.229} C_VEL
LIN {X 0,Y 374.527,Z 399.546,A -85,B 0,C 180,E1 -12334.306,E2 -12334.306} C_VEL
LIN {X 0,Y 374.567,Z 396.536,A -85,B 0,C 180,E1 -12336.044,E2 -12336.044} C_VEL
LIN {X 0,Y 374.823,Z 392.974,A -85,B 0,C 180,E1 -12337.543,E2 -12337.543} C_VEL
LIN {X 0,Y 375.204,Z 388.015,A -85,B 0,C 180,E1 -12339.162,E2 -12339.162} C_VEL
LIN {X 0,Y 375.79,Z 381.767,A -85,B 0,C 180,E1 -12340.78,E2 -12340.78} C_VEL
LIN {X 0,Y 376.599,Z 374.029,A -85,B 0,C 180,E1 -12342.394,E2 -12342.394} C_VEL
LIN {X 0,Y 377.52,Z 366.154,A -85,B 0,C 180,E1 -12343.731,E2 -12343.731} C_VEL
LIN {X 0,Y 378.372,Z 356.58,A -85,B 0,C 180,E1 -12345.073,E2 -12345.073} C_VEL
LIN {X 0,Y 379.504,Z 346.007,A -85,B 0,C 180,E1 -12346.267,E2 -12346.267} C_VEL
LIN {X 0,Y 380.701,Z 334.311,A -85,B 0,C 180,E1 -12347.319,E2 -12347.319} C_VEL
LIN {X 0,Y 381.716,Z 321.981,A -85,B 0,C 180,E1 -12348.171,E2 -12348.171} C_VEL
LIN {X 0,Y 382.646,Z 308.58,A -85,B 0,C 180,E1 -12348.854,E2 -12348.854} C_VEL
LIN {X 0,Y 383.362,Z 294.922,A -85,B 0,C 180,E1 -12349.304,E2 -12349.304} C_VEL
LIN {X 0,Y 385.124,Z 220.581,A -85,B 0,C 180,E1 -12350.999,E2 -12350.999} C_VEL
LIN {X 0,Y 382.092,Z 201.782,A -85,B 0,C 180,E1 -12351.7,E2 -12351.7} C_VEL
LIN {X 0,Y 379.266,Z 188.65,A -85,B 0,C 180,E1 -12352.273,E2 -12352.273} C_VEL
LIN {X 0,Y 380.307,Z 178.525,A -85,B 0,C 180,E1 -12354.529,E2 -12354.529} C_VEL
LIN {X 0,Y 379.978,Z 174.622,A -85,B 0,C 180,E1 -12355.47,E2 -12355.47} C_VEL
LIN {X 0,Y 377.701,Z 163.763,A -85,B 0,C 180,E1 -12358.285,E2 -12358.285} C_VEL
LIN {X 0,Y 375.977,Z 156.653,A -85,B 0,C 180,E1 -12360.274,E2 -12360.274} C_VEL
LIN {X 0,Y 375.96,Z 156.653,A -85,B 0,C 180,E1 -12364.112,E2 -12364.112} C_VEL
LIN {X 0,Y 375.95,Z 156.658,A -85,B 0,C 180,E1 -12366.742,E2 -12366.742} C_VEL
LIN {X 0,Y 375.941,Z 156.655,A -85,B 0,C 180,E1 -12369.962,E2 -12369.962} C_VEL
LIN {X 0,Y 375.928,Z 156.653,A -85,B 0,C 180,E1 -12373.767,E2 -12373.767} C_VEL
LIN {X 0,Y 375.935,Z 156.65,A -85,B 0,C 180,E1 -12376.812,E2 -12376.812} C_VEL
LIN {X 0,Y 375.937,Z 156.655,A -85,B 0,C 180,E1 -12380.534,E2 -12380.534} C_VEL
LIN {X 0,Y 375.961,Z 156.649,A -85,B 0,C 180,E1 -12383.497,E2 -12383.497} C_VEL
LIN {X 0,Y 375.961,Z 156.653,A -85,B 0,C 180,E1 -12385.889,E2 -12385.889} C_VEL
LIN {X 0,Y 375.964,Z 156.649,A -85,B 0,C 180,E1 -12389.687,E2 -12389.687} C_VEL
LIN {X 0,Y 375.92,Z 156.655,A -85,B 0,C 180,E1 -12392.135,E2 -12392.135} C_VEL
LIN {X 0,Y 375.962,Z 156.652,A -85,B 0,C 180,E1 -12395.716,E2 -12395.716} C_VEL
LIN {X 0,Y 375.984,Z 156.645,A -85,B 0,C 180,E1 -12399.197,E2 -12399.197} C_VEL
LIN {X 0,Y 376.014,Z 156.648,A -85,B 0,C 180,E1 -12402.599,E2 -12402.599} C_VEL
LIN {X 0,Y 376.094,Z 156.637,A -85,B 0,C 180,E1 -12406.343,E2 -12406.343} C_VEL
LIN {X 0,Y 376.117,Z 156.637,A -85,B 0,C 180,E1 -12410.319,E2 -12410.319} C_VEL
LIN {X 0,Y 376.202,Z 156.626,A -85,B 0,C 180,E1 -12413.564,E2 -12413.564} C_VEL
LIN {X 0,Y 376.342,Z 156.608,A -85,B 0,C 180,E1 -12417.86,E2 -12417.86} C_VEL
LIN {X 0,Y 376.31,Z 156.659,A -85,B 0,C 180,E1 -12421.739,E2 -12421.739} C_VEL
LIN {X 0,Y 379.175,Z 169.717,A -85,B 0,C 180,E1 -12425.318,E2 -12425.318} C_VEL
LIN {X 0,Y 379.532,Z 171.71,A -85,B 0,C 180,E1 -12425.812,E2 -12425.812} C_VEL
LIN {X 0,Y 381.712,Z 177.772,A -85,B 0,C 180,E1 -12426.149,E2 -12426.149} C_VEL
LIN {X 0,Y 384.975,Z 191.904,A -85,B 0,C 180,E1 -12426.76,E2 -12426.76} C_VEL
LIN {X 0,Y 385.829,Z 197.476,A -85,B 0,C 180,E1 -12426.964,E2 -12426.964} C_VEL
LIN {X 0,Y 383.43,Z 280.73,A -85,B 0,C 180,E1 -12428.877,E2 -12428.877} C_VEL
LIN {X 0,Y 382.805,Z 293.329,A -85,B 0,C 180,E1 -12429.364,E2 -12429.364} C_VEL
LIN {X 0,Y 382.042,Z 305.906,A -85,B 0,C 180,E1 -12430.065,E2 -12430.065} C_VEL
LIN {X 0,Y 381.057,Z 318.51,A -85,B 0,C 180,E1 -12431.015,E2 -12431.015} C_VEL
LIN {X 0,Y 379.988,Z 330.167,A -85,B 0,C 180,E1 -12432.145,E2 -12432.145} C_VEL
LIN {X 0,Y 378.834,Z 340.505,A -85,B 0,C 180,E1 -12433.409,E2 -12433.409} C_VEL
LIN {X 0,Y 377.814,Z 349.933,A -85,B 0,C 180,E1 -12434.839,E2 -12434.839} C_VEL
LIN {X 0,Y 376.971,Z 357.468,A -85,B 0,C 180,E1 -12436.24,E2 -12436.24} C_VEL
LIN {X 0,Y 376.245,Z 363.906,A -85,B 0,C 180,E1 -12437.701,E2 -12437.701} C_VEL
LIN {X 0,Y 375.654,Z 368.992,A -85,B 0,C 180,E1 -12439.112,E2 -12439.112} C_VEL
LIN {X 0,Y 375.196,Z 373.958,A -85,B 0,C 180,E1 -12440.849,E2 -12440.849} C_VEL
LIN {X 0,Y 374.822,Z 377.653,A -85,B 0,C 180,E1 -12442.606,E2 -12442.606} C_VEL
LIN {X 0,Y 374.519,Z 380.175,A -85,B 0,C 180,E1 -12444.384,E2 -12444.384} C_VEL
LIN {X 0,Y 374.396,Z 381.315,A -85,B 0,C 180,E1 -12445.704,E2 -12445.704} C_VEL
LIN {X 0,Y 374.32,Z 381.764,A -85,B 0,C 180,E1 -12446.783,E2 -12446.783} C_VEL
LIN {X 0,Y 374.31,Z 381.75,A -85,B 0,C 180,E1 -12448.057,E2 -12448.057} C_VEL
LIN {X 0,Y 374.294,Z 381.262,A -85,B 0,C 180,E1 -12449.222,E2 -12449.222} C_VEL
LIN {X 0,Y 374.376,Z 380.163,A -85,B 0,C 180,E1 -12450.455,E2 -12450.455} C_VEL
LIN {X 0,Y 374.564,Z 377.343,A -85,B 0,C 180,E1 -12452.397,E2 -12452.397} C_VEL
LIN {X 0,Y 374.8,Z 372.843,A -85,B 0,C 180,E1 -12454.404,E2 -12454.404} C_VEL
LIN {X 0,Y 375.219,Z 366.801,A -85,B 0,C 180,E1 -12456.349,E2 -12456.349} C_VEL
LIN {X 0,Y 375.739,Z 359.611,A -85,B 0,C 180,E1 -12458.116,E2 -12458.116} C_VEL
LIN {X 0,Y 376.354,Z 351.205,A -85,B 0,C 180,E1 -12459.752,E2 -12459.752} C_VEL
LIN {X 0,Y 377.04,Z 342.832,A -85,B 0,C 180,E1 -12461.076,E2 -12461.076} C_VEL
LIN {X 0,Y 377.771,Z 332.494,A -85,B 0,C 180,E1 -12462.407,E2 -12462.407} C_VEL
LIN {X 0,Y 378.662,Z 320.571,A -85,B 0,C 180,E1 -12463.626,E2 -12463.626} C_VEL
LIN {X 0,Y 379.499,Z 308.827,A -85,B 0,C 180,E1 -12464.562,E2 -12464.562} C_VEL
LIN {X 0,Y 380.074,Z 297.068,A -85,B 0,C 180,E1 -12465.281,E2 -12465.281} C_VEL
LIN {X 0,Y 380.574,Z 283.94,A -85,B 0,C 180,E1 -12465.862,E2 -12465.862} C_VEL
LIN {X 0,Y 380.984,Z 270.875,A -85,B 0,C 180,E1 -12466.223,E2 -12466.223} C_VEL
LIN {X 0,Y 382.391,Z 194.48,A -85,B 0,C 180,E1 -12467.867,E2 -12467.867} C_VEL
LIN {X 0,Y 378.175,Z 170.542,A -85,B 0,C 180,E1 -12468.631,E2 -12468.631} C_VEL
LIN {X 0,Y 377.86,Z 166.376,A -85,B 0,C 180,E1 -12469.693,E2 -12469.693} C_VEL
LIN {X 0,Y 375.993,Z 156.651,A -85,B 0,C 180,E1 -12472.338,E2 -12472.338} C_VEL
LIN {X 0,Y 375.964,Z 156.651,A -85,B 0,C 180,E1 -12475.888,E2 -12475.888} C_VEL
LIN {X 0,Y 375.965,Z 156.65,A -85,B 0,C 180,E1 -12479.687,E2 -12479.687} C_VEL
LIN {X 0,Y 375.921,Z 156.659,A -85,B 0,C 180,E1 -12482.134,E2 -12482.134} C_VEL
LIN {X 0,Y 375.941,Z 156.657,A -85,B 0,C 180,E1 -12484.533,E2 -12484.533} C_VEL
LIN {X 0,Y 375.975,Z 156.649,A -85,B 0,C 180,E1 -12486.886,E2 -12486.886} C_VEL
LIN {X 0,Y 375.967,Z 156.655,A -85,B 0,C 180,E1 -12490.337,E2 -12490.337} C_VEL
LIN {X 0,Y 375.966,Z 156.652,A -85,B 0,C 180,E1 -12493.715,E2 -12493.715} C_VEL
LIN {X 0,Y 376.107,Z 156.632,A -85,B 0,C 180,E1 -12497.041,E2 -12497.041} C_VEL
LIN {X 0,Y 376.112,Z 156.634,A -85,B 0,C 180,E1 -12500.317,E2 -12500.317} C_VEL
LIN {X 0,Y 376.198,Z 156.623,A -85,B 0,C 180,E1 -12503.563,E2 -12503.563} C_VEL
LIN {X 0,Y 376.341,Z 156.609,A -85,B 0,C 180,E1 -12507.859,E2 -12507.859} C_VEL
LIN {X 0,Y 376.341,Z 156.605,A -85,B 0,C 180,E1 -12512.14,E2 -12512.14} C_VEL
LIN {X 0,Y 376.27,Z 156.612,A -85,B 0,C 180,E1 -12512.443,E2 -12512.443} C_VEL
LIN {X 0,Y 375.477,Z 156.715,A -85,B 0,C 180,E1 -12513.335,E2 -12513.335} C_VEL
LIN {X 0,Y 372.589,Z 157.07,A -85,B 0,C 180,E1 -12514.788,E2 -12514.788} C_VEL
LIN {X 0,Y 370.218,Z 157.369,A -85,B 0,C 180,E1 -12515.962,E2 -12515.962} C_VEL
LIN {X 0,Y 369.204,Z 157.492,A -85,B 0,C 180,E1 -12516.87,E2 -12516.87} C_VEL
LIN {X 0,Y 369.118,Z 157.504,A -85,B 0,C 180,E1 -12517.177,E2 -12517.177} C_VEL
LIN {X 0,Y 369.061,Z 157.513,A -85,B 0,C 180,E1 -12519.867,E2 -12519.867} C_VEL
LIN {X 0,Y 369.04,Z 157.516,A -85,B 0,C 180,E1 -12523.771,E2 -12523.771} C_VEL
LIN {X 0,Y 368.955,Z 157.526,A -85,B 0,C 180,E1 -12527.744,E2 -12527.744} C_VEL
LIN {X 0,Y 368.91,Z 157.533,A -85,B 0,C 180,E1 -12531.22,E2 -12531.22} C_VEL
LIN {X 0,Y 368.908,Z 157.53,A -85,B 0,C 180,E1 -12533.873,E2 -12533.873} C_VEL
LIN {X 0,Y 368.857,Z 157.541,A -85,B 0,C 180,E1 -12537.211,E2 -12537.211} C_VEL
LIN {X 0,Y 368.892,Z 157.532,A -85,B 0,C 180,E1 -12539.691,E2 -12539.691} C_VEL
LIN {X 0,Y 368.894,Z 157.536,A -85,B 0,C 180,E1 -12543.041,E2 -12543.041} C_VEL
LIN {X 0,Y 368.91,Z 157.528,A -85,B 0,C 180,E1 -12546.196,E2 -12546.196} C_VEL
LIN {X 0,Y 368.873,Z 157.539,A -85,B 0,C 180,E1 -12548.956,E2 -12548.956} C_VEL
LIN {X 0,Y 368.867,Z 157.534,A -85,B 0,C 180,E1 -12552.006,E2 -12552.006} C_VEL
LIN {X 0,Y 368.871,Z 157.537,A -85,B 0,C 180,E1 -12555.174,E2 -12555.174} C_VEL
LIN {X 0,Y 368.861,Z 157.535,A -85,B 0,C 180,E1 -12558.174,E2 -12558.174} C_VEL
LIN {X 0,Y 368.872,Z 157.534,A -85,B 0,C 180,E1 -12561.365,E2 -12561.365} C_VEL
LIN {X 0,Y 368.931,Z 157.528,A -85,B 0,C 180,E1 -12565.145,E2 -12565.145} C_VEL
LIN {X 0,Y 368.908,Z 157.531,A -85,B 0,C 180,E1 -12569.044,E2 -12569.044} C_VEL
LIN {X 0,Y 368.901,Z 157.529,A -85,B 0,C 180,E1 -12571.557,E2 -12571.557} C_VEL
LIN {X 0,Y 368.913,Z 157.53,A -85,B 0,C 180,E1 -12574.013,E2 -12574.013} C_VEL
LIN {X 0,Y 368.89,Z 157.531,A -85,B 0,C 180,E1 -12577.602,E2 -12577.602} C_VEL
LIN {X 0,Y 368.913,Z 157.528,A -85,B 0,C 180,E1 -12581.103,E2 -12581.103} C_VEL
LIN {X 0,Y 368.933,Z 157.529,A -85,B 0,C 180,E1 -12584.532,E2 -12584.532} C_VEL
LIN {X 0,Y 369.05,Z 157.512,A -85,B 0,C 180,E1 -12586.79,E2 -12586.79} C_VEL
LIN {X 0,Y 369.05,Z 157.517,A -85,B 0,C 180,E1 -12590.131,E2 -12590.131} C_VEL
LIN {X 0,Y 369.151,Z 157.499,A -85,B 0,C 180,E1 -12593.441,E2 -12593.441} C_VEL
LIN {X 0,Y 369.293,Z 157.485,A -85,B 0,C 180,E1 -12597.818,E2 -12597.818} C_VEL
LIN {X 0,Y 369.194,Z 157.493,A -85,B 0,C 180,E1 -12601.091,E2 -12601.091} C_VEL
LIN {X 0,Y 369.293,Z 157.484,A -85,B 0,C 180,E1 -12602.181,E2 -12602.181} C_VEL
LIN {X 0,Y 369.15,Z 157.499,A -85,B 0,C 180,E1 -12606.559,E2 -12606.559} C_VEL
LIN {X 0,Y 369.05,Z 157.516,A -85,B 0,C 180,E1 -12609.869,E2 -12609.869} C_VEL
LIN {X 0,Y 369.03,Z 157.519,A -85,B 0,C 180,E1 -12613.772,E2 -12613.772} C_VEL
LIN {X 0,Y 368.946,Z 157.529,A -85,B 0,C 180,E1 -12617.745,E2 -12617.745} C_VEL
LIN {X 0,Y 368.901,Z 157.533,A -85,B 0,C 180,E1 -12621.221,E2 -12621.221} C_VEL
LIN {X 0,Y 368.9,Z 157.532,A -85,B 0,C 180,E1 -12623.874,E2 -12623.874} C_VEL
LIN {X 0,Y 368.849,Z 157.541,A -85,B 0,C 180,E1 -12627.212,E2 -12627.212} C_VEL
LIN {X 0,Y 368.884,Z 157.534,A -85,B 0,C 180,E1 -12629.693,E2 -12629.693} C_VEL
LIN {X 0,Y 368.889,Z 157.535,A -85,B 0,C 180,E1 -12633.043,E2 -12633.043} C_VEL
LIN {X 0,Y 368.904,Z 157.529,A -85,B 0,C 180,E1 -12636.198,E2 -12636.198} C_VEL
LIN {X 0,Y 368.867,Z 157.538,A -85,B 0,C 180,E1 -12638.958,E2 -12638.958} C_VEL
LIN {X 0,Y 368.852,Z 157.536,A -85,B 0,C 180,E1 -12642.006,E2 -12642.006} C_VEL
LIN {X 0,Y 368.868,Z 157.538,A -85,B 0,C 180,E1 -12645.176,E2 -12645.176} C_VEL
LIN {X 0,Y 368.855,Z 157.536,A -85,B 0,C 180,E1 -12648.175,E2 -12648.175} C_VEL
LIN {X 0,Y 368.871,Z 157.535,A -85,B 0,C 180,E1 -12651.367,E2 -12651.367} C_VEL
LIN {X 0,Y 368.926,Z 157.529,A -85,B 0,C 180,E1 -12655.147,E2 -12655.147} C_VEL
LIN {X 0,Y 368.892,Z 157.535,A -85,B 0,C 180,E1 -12659.044,E2 -12659.044} C_VEL
LIN {X 0,Y 368.926,Z 157.619,A -85,B 0,C 180,E1 -12661.285,E2 -12661.285} C_VEL
LIN {X 0,Y 371.452,Z 170.44,A -85,B 0,C 180,E1 -12664.481,E2 -12664.481} C_VEL
LIN {X 0,Y 372.116,Z 175.716,A -85,B 0,C 180,E1 -12665.747,E2 -12665.747} C_VEL
LIN {X 0,Y 371.31,Z 185.824,A -85,B 0,C 180,E1 -12668.041,E2 -12668.041} C_VEL
LIN {X 0,Y 370.949,Z 190.675,A -85,B 0,C 180,E1 -12669.084,E2 -12669.084} C_VEL
LIN {X 0,Y 375.309,Z 221.906,A -85,B 0,C 180,E1 -12670.011,E2 -12670.011} C_VEL
LIN {X 0,Y 373.753,Z 299.508,A -85,B 0,C 180,E1 -12671.749,E2 -12671.749} C_VEL
LIN {X 0,Y 373.094,Z 313.365,A -85,B 0,C 180,E1 -12672.283,E2 -12672.283} C_VEL
LIN {X 0,Y 372.355,Z 325.862,A -85,B 0,C 180,E1 -12672.99,E2 -12672.99} C_VEL
LIN {X 0,Y 371.515,Z 338.317,A -85,B 0,C 180,E1 -12673.94,E2 -12673.94} C_VEL
LIN {X 0,Y 370.712,Z 348.968,A -85,B 0,C 180,E1 -12674.972,E2 -12674.972} C_VEL
LIN {X 0,Y 369.954,Z 359.611,A -85,B 0,C 180,E1 -12676.264,E2 -12676.264} C_VEL
LIN {X 0,Y 369.171,Z 368.766,A -85,B 0,C 180,E1 -12677.634,E2 -12677.634} C_VEL
LIN {X 0,Y 368.396,Z 377.695,A -85,B 0,C 180,E1 -12679.281,E2 -12679.281} C_VEL
LIN {X 0,Y 367.97,Z 384.799,A -85,B 0,C 180,E1 -12680.935,E2 -12680.935} C_VEL
LIN {X 0,Y 367.654,Z 391.293,A -85,B 0,C 180,E1 -12682.863,E2 -12682.863} C_VEL
LIN {X 0,Y 367.457,Z 395.513,A -85,B 0,C 180,E1 -12684.513,E2 -12684.513} C_VEL
LIN {X 0,Y 367.474,Z 397.71,A -85,B 0,C 180,E1 -12685.614,E2 -12685.614} C_VEL
LIN {X 0,Y 367.383,Z 399.415,A -85,B 0,C 180,E1 -12686.711,E2 -12686.711} C_VEL
LIN {X 0,Y 367.376,Z 400.703,A -85,B 0,C 180,E1 -12687.808,E2 -12687.808} C_VEL
LIN {X 0,Y 367.421,Z 401.571,A -85,B 0,C 180,E1 -12688.905,E2 -12688.905} C_VEL
LIN {X 0,Y 367.457,Z 401.975,A -85,B 0,C 180,E1 -12690.001,E2 -12690.001} C_VEL
LIN {X 0,Y 367.403,Z 401.967,A -85,B 0,C 180,E1 -12691.097,E2 -12691.097} C_VEL
LIN {X 0,Y 367.357,Z 401.554,A -85,B 0,C 180,E1 -12692.194,E2 -12692.194} C_VEL
LIN {X 0,Y 367.377,Z 400.724,A -85,B 0,C 180,E1 -12693.291,E2 -12693.291} C_VEL
LIN {X 0,Y 367.435,Z 399.436,A -85,B 0,C 180,E1 -12694.389,E2 -12694.389} C_VEL
LIN {X 0,Y 367.474,Z 396.776,A -85,B 0,C 180,E1 -12696.007,E2 -12696.007} C_VEL
LIN {X 0,Y 367.75,Z 392.937,A -85,B 0,C 180,E1 -12697.689,E2 -12697.689} C_VEL
LIN {X 0,Y 368.188,Z 388.039,A -85,B 0,C 180,E1 -12699.338,E2 -12699.338} C_VEL
LIN {X 0,Y 368.892,Z 380.716,A -85,B 0,C 180,E1 -12701.262,E2 -12701.262} C_VEL
LIN {X 0,Y 369.678,Z 374.196,A -85,B 0,C 180,E1 -12702.629,E2 -12702.629} C_VEL
LIN {X 0,Y 370.63,Z 366.393,A -85,B 0,C 180,E1 -12703.992,E2 -12703.992} C_VEL
LIN {X 0,Y 371.651,Z 355.858,A -85,B 0,C 180,E1 -12705.493,E2 -12705.493} C_VEL
LIN {X 0,Y 372.874,Z 345.171,A -85,B 0,C 180,E1 -12706.705,E2 -12706.705} C_VEL
LIN {X 0,Y 374.154,Z 333.263,A -85,B 0,C 180,E1 -12707.773,E2 -12707.773} C_VEL
LIN {X 0,Y 375.301,Z 319.666,A -85,B 0,C 180,E1 -12708.705,E2 -12708.705} C_VEL
LIN {X 0,Y 376.246,Z 306.988,A -85,B 0,C 180,E1 -12709.329,E2 -12709.329} C_VEL
LIN {X 0,Y 376.947,Z 292.69,A -85,B 0,C 180,E1 -12709.787,E2 -12709.787} C_VEL
LIN {X 0,Y 378.743,Z 221.592,A -85,B 0,C 180,E1 -12711.447,E2 -12711.447} C_VEL
LIN {X 0,Y 375.541,Z 201.735,A -85,B 0,C 180,E1 -12712.213,E2 -12712.213} C_VEL
LIN {X 0,Y 372.597,Z 188.337,A -85,B 0,C 180,E1 -12712.848,E2 -12712.848} C_VEL
LIN {X 0,Y 373.523,Z 179.332,A -85,B 0,C 180,E1 -12714.903,E2 -12714.903} C_VEL
LIN {X 0,Y 372.147,Z 171.368,A -85,B 0,C 180,E1 -12716.953,E2 -12716.953} C_VEL
LIN {X 0,Y 370.025,Z 161.688,A -85,B 0,C 180,E1 -12719.593,E2 -12719.593} C_VEL
LIN {X 0,Y 368.92,Z 157.533,A -85,B 0,C 180,E1 -12720.841,E2 -12720.841} C_VEL
LIN {X 0,Y 368.933,Z 157.533,A -85,B 0,C 180,E1 -12724.855,E2 -12724.855} C_VEL
LIN {X 0,Y 368.878,Z 157.538,A -85,B 0,C 180,E1 -12728.634,E2 -12728.634} C_VEL
LIN {X 0,Y 368.867,Z 157.535,A -85,B 0,C 180,E1 -12732.007,E2 -12732.007} C_VEL
LIN {X 0,Y 368.877,Z 157.533,A -85,B 0,C 180,E1 -12735.175,E2 -12735.175} C_VEL
LIN {X 0,Y 368.872,Z 157.532,A -85,B 0,C 180,E1 -12738.176,E2 -12738.176} C_VEL
LIN {X 0,Y 368.879,Z 157.529,A -85,B 0,C 180,E1 -12741.367,E2 -12741.367} C_VEL
LIN {X 0,Y 368.934,Z 157.529,A -85,B 0,C 180,E1 -12745.146,E2 -12745.146} C_VEL
LIN {X 0,Y 368.916,Z 157.526,A -85,B 0,C 180,E1 -12749.045,E2 -12749.045} C_VEL
LIN {X 0,Y 368.91,Z 157.527,A -85,B 0,C 180,E1 -12751.558,E2 -12751.558} C_VEL
LIN {X 0,Y 368.901,Z 157.53,A -85,B 0,C 180,E1 -12755.221,E2 -12755.221} C_VEL
LIN {X 0,Y 368.902,Z 157.529,A -85,B 0,C 180,E1 -12757.603,E2 -12757.603} C_VEL
LIN {X 0,Y 368.93,Z 157.527,A -85,B 0,C 180,E1 -12761.105,E2 -12761.105} C_VEL
LIN {X 0,Y 368.944,Z 157.529,A -85,B 0,C 180,E1 -12764.533,E2 -12764.533} C_VEL
LIN {X 0,Y 369.062,Z 157.514,A -85,B 0,C 180,E1 -12766.791,E2 -12766.791} C_VEL
LIN {X 0,Y 369.067,Z 157.514,A -85,B 0,C 180,E1 -12770.132,E2 -12770.132} C_VEL
LIN {X 0,Y 369.163,Z 157.503,A -85,B 0,C 180,E1 -12773.441,E2 -12773.441} C_VEL
LIN {X 0,Y 369.306,Z 157.484,A -85,B 0,C 180,E1 -12777.819,E2 -12777.819} C_VEL
LIN {X 0,Y 369.219,Z 157.611,A -85,B 0,C 180,E1 -12781.193,E2 -12781.193} C_VEL
LIN {X 0,Y 370.524,Z 162.848,A -85,B 0,C 180,E1 -12782.718,E2 -12782.718} C_VEL
LIN {X 0,Y 372.493,Z 172.002,A -85,B 0,C 180,E1 -12785.227,E2 -12785.227} C_VEL
LIN {X 0,Y 375.676,Z 180.187,A -85,B 0,C 180,E1 -12785.72,E2 -12785.72} C_VEL
LIN {X 0,Y 379.034,Z 195.139,A -85,B 0,C 180,E1 -12786.388,E2 -12786.388} C_VEL
LIN {X 0,Y 379.474,Z 198.332,A -85,B 0,C 180,E1 -12786.504,E2 -12786.504} C_VEL
LIN {X 0,Y 376.941,Z 280.404,A -85,B 0,C 180,E1 -12788.426,E2 -12788.426} C_VEL
LIN {X 0,Y 376.274,Z 293.986,A -85,B 0,C 180,E1 -12788.965,E2 -12788.965} C_VEL
LIN {X 0,Y 375.424,Z 306.701,A -85,B 0,C 180,E1 -12789.7,E2 -12789.7} C_VEL
LIN {X 0,Y 374.363,Z 319.349,A -85,B 0,C 180,E1 -12790.684,E2 -12790.684} C_VEL
LIN {X 0,Y 373.307,Z 330.284,A -85,B 0,C 180,E1 -12791.769,E2 -12791.769} C_VEL
LIN {X 0,Y 372.057,Z 340.991,A -85,B 0,C 180,E1 -12793.102,E2 -12793.102} C_VEL
LIN {X 0,Y 370.985,Z 350.262,A -85,B 0,C 180,E1 -12794.535,E2 -12794.535} C_VEL
LIN {X 0,Y 370.077,Z 357.893,A -85,B 0,C 180,E1 -12795.984,E2 -12795.984} C_VEL
LIN {X 0,Y 369.115,Z 365.592,A -85,B 0,C 180,E1 -12797.821,E2 -12797.821} C_VEL
LIN {X 0,Y 368.464,Z 371.118,A -85,B 0,C 180,E1 -12799.499,E2 -12799.499} C_VEL
LIN {X 0,Y 368.014,Z 375.612,A -85,B 0,C 180,E1 -12801.275,E2 -12801.275} C_VEL
LIN {X 0,Y 367.759,Z 377.921,A -85,B 0,C 180,E1 -12802.471,E2 -12802.471} C_VEL
LIN {X 0,Y 367.539,Z 379.714,A -85,B 0,C 180,E1 -12803.676,E2 -12803.676} C_VEL
LIN {X 0,Y 367.364,Z 381.018,A -85,B 0,C 180,E1 -12804.891,E2 -12804.891} C_VEL
LIN {X 0,Y 367.265,Z 381.768,A -85,B 0,C 180,E1 -12806.113,E2 -12806.113} C_VEL
LIN {X 0,Y 367.196,Z 382.046,A -85,B 0,C 180,E1 -12807.346,E2 -12807.346} C_VEL
LIN {X 0,Y 367.206,Z 381.753,A -85,B 0,C 180,E1 -12808.587,E2 -12808.587} C_VEL
LIN {X 0,Y 367.281,Z 380.216,A -85,B 0,C 180,E1 -12810.56,E2 -12810.56} C_VEL
LIN {X 0,Y 367.517,Z 376.968,A -85,B 0,C 180,E1 -12812.71,E2 -12812.71} C_VEL
LIN {X 0,Y 367.698,Z 373.682,A -85,B 0,C 180,E1 -12814.203,E2 -12814.203} C_VEL
LIN {X 0,Y 368.013,Z 368.572,A -85,B 0,C 180,E1 -12815.962,E2 -12815.962} C_VEL
LIN {X 0,Y 368.585,Z 361.385,A -85,B 0,C 180,E1 -12817.864,E2 -12817.864} C_VEL
LIN {X 0,Y 369.094,Z 354.692,A -85,B 0,C 180,E1 -12819.281,E2 -12819.281} C_VEL
LIN {X 0,Y 369.844,Z 345.588,A -85,B 0,C 180,E1 -12820.851,E2 -12820.851} C_VEL
LIN {X 0,Y 370.632,Z 335.046,A -85,B 0,C 180,E1 -12822.308,E2 -12822.308} C_VEL
LIN {X 0,Y 371.461,Z 324.39,A -85,B 0,C 180,E1 -12823.489,E2 -12823.489} C_VEL
LIN {X 0,Y 372.351,Z 311.803,A -85,B 0,C 180,E1 -12824.58,E2 -12824.58} C_VEL
LIN {X 0,Y 373.08,Z 299.061,A -85,B 0,C 180,E1 -12825.423,E2 -12825.423} C_VEL
LIN {X 0,Y 373.622,Z 285.042,A -85,B 0,C 180,E1 -12826.077,E2 -12826.077} C_VEL
LIN {X 0,Y 374.079,Z 272.497,A -85,B 0,C 180,E1 -12826.448,E2 -12826.448} C_VEL
LIN {X 0,Y 375.557,Z 195.166,A -85,B 0,C 180,E1 -12828.154,E2 -12828.154} C_VEL
LIN {X 0,Y 371.217,Z 170.783,A -85,B 0,C 180,E1 -12828.938,E2 -12828.938} C_VEL
LIN {X 0,Y 370.331,Z 164.802,A -85,B 0,C 180,E1 -12830.523,E2 -12830.523} C_VEL
LIN {X 0,Y 368.938,Z 157.531,A -85,B 0,C 180,E1 -12832.54,E2 -12832.54} C_VEL
LIN {X 0,Y 368.941,Z 157.526,A -85,B 0,C 180,E1 -12835.146,E2 -12835.146} C_VEL
LIN {X 0,Y 368.901,Z 157.531,A -85,B 0,C 180,E1 -12839.043,E2 -12839.043} C_VEL
LIN {X 0,Y 368.912,Z 157.528,A -85,B 0,C 180,E1 -12841.557,E2 -12841.557} C_VEL
LIN {X 0,Y 368.924,Z 157.53,A -85,B 0,C 180,E1 -12844.013,E2 -12844.013} C_VEL
LIN {X 0,Y 368.9,Z 157.53,A -85,B 0,C 180,E1 -12847.602,E2 -12847.602} C_VEL
LIN {X 0,Y 368.907,Z 157.529,A -85,B 0,C 180,E1 -12851.102,E2 -12851.102} C_VEL
LIN {X 0,Y 368.939,Z 157.527,A -85,B 0,C 180,E1 -12854.532,E2 -12854.532} C_VEL
LIN {X 0,Y 369.062,Z 157.51,A -85,B 0,C 180,E1 -12856.789,E2 -12856.789} C_VEL
LIN {X 0,Y 369.063,Z 157.515,A -85,B 0,C 180,E1 -12860.131,E2 -12860.131} C_VEL
LIN {X 0,Y 369.159,Z 157.499,A -85,B 0,C 180,E1 -12863.44,E2 -12863.44} C_VEL
LIN {X 0,Y 369.305,Z 157.485,A -85,B 0,C 180,E1 -12867.818,E2 -12867.818} C_VEL
LIN {X 0,Y 369.305,Z 157.481,A -85,B 0,C 180,E1 -12872.18,E2 -12872.18} C_VEL
LIN {X 0,Y 369.156,Z 157.498,A -85,B 0,C 180,E1 -12876.558,E2 -12876.558} C_VEL
LIN {X 0,Y 369.118,Z 157.504,A -85,B 0,C 180,E1 -12877.177,E2 -12877.177} C_VEL
LIN {X 0,Y 368.426,Z 157.595,A -85,B 0,C 180,E1 -12878.087,E2 -12878.087} C_VEL
LIN {X 0,Y 365.512,Z 157.958,A -85,B 0,C 180,E1 -12879.566,E2 -12879.566} C_VEL
LIN {X 0,Y 363.061,Z 158.258,A -85,B 0,C 180,E1 -12880.762,E2 -12880.762} C_VEL
LIN {X 0,Y 362.023,Z 158.391,A -85,B 0,C 180,E1 -12881.689,E2 -12881.689} C_VEL
LIN {X 0,Y 361.945,Z 158.395,A -85,B 0,C 180,E1 -12882.003,E2 -12882.003} C_VEL
LIN {X 0,Y 361.936,Z 158.397,A -85,B 0,C 180,E1 -12884.62,E2 -12884.62} C_VEL
LIN {X 0,Y 361.885,Z 158.404,A -85,B 0,C 180,E1 -12888.102,E2 -12888.102} C_VEL
LIN {X 0,Y 361.854,Z 158.411,A -85,B 0,C 180,E1 -12891.654,E2 -12891.654} C_VEL
LIN {X 0,Y 361.86,Z 158.413,A -85,B 0,C 180,E1 -12895.294,E2 -12895.294} C_VEL
LIN {X 0,Y 361.855,Z 158.412,A -85,B 0,C 180,E1 -12899.072,E2 -12899.072} C_VEL
LIN {X 0,Y 361.846,Z 158.413,A -85,B 0,C 180,E1 -12902.944,E2 -12902.944} C_VEL
LIN {X 0,Y 361.862,Z 158.408,A -85,B 0,C 180,E1 -12905.636,E2 -12905.636} C_VEL
LIN {X 0,Y 361.824,Z 158.417,A -85,B 0,C 180,E1 -12909.017,E2 -12909.017} C_VEL
